// TwinCAT 3 PLC project SIM_1
// ProgramVersion: 3.1.4026.25
// libraries:
//   OC_Core, * (Open Commissioning)
//   Tc2_Math, * (Beckhoff Automation GmbH)
//   Tc2_Standard, * (Beckhoff Automation GmbH)
//   Tc2_System, * (Beckhoff Automation GmbH)
//   Tc2_Utilities, * (Beckhoff Automation GmbH)
//   Tc3_Module, * (Beckhoff Automation GmbH)
// project tree:
//   FG_01/ FG_01.TcPOU
//   FG_02/ FG_02.TcPOU
//   FG_03/ FG_03.TcPOU
//   FG_04/ FG_04.TcPOU
//   FG_05/ FG_05.TcPOU
//   FG_System/ FG_System.TcPOU
//   FG_Transport/ FG_Transport.TcPOU
//   Library/ FB_Camera.TcPOU
//   / MAIN.TcPOU (not stored), PlcTask.TcTTO
//   Sil/PLC/ GVL_PLC.TcGVL, ST_PLCInputs.TcDUT, ST_PLCOutputs.TcDUT
// real-time tasks:
//   TASK PlcTask: cycle T#1ms, priority 4, ADS port 350

CONFIGURATION SIM_1
    RESOURCE PLC ON TwinCAT3
        TASK PlcTask(INTERVAL := T#1ms, PRIORITY := 4);
        PROGRAM MAIN WITH PlcTask : MAIN;
    END_RESOURCE
END_CONFIGURATION

// ---- Sil/PLC/ST_PLCInputs.TcDUT
{attribute 'pack_mode' := '0'}
TYPE ST_PLCInputs :
STRUCT
	I0: BYTE;
	I1: BYTE;
	I2: BYTE;
	I3: BYTE;
	I4: BYTE;
	I5: BYTE;
	I6: BYTE;
	I7: BYTE;
	I8: BYTE;
	I9: BYTE;
	I10: BYTE;
	I11: BYTE;
	I12: BYTE;
	I13: BYTE;
	I14: BYTE;
	I15: BYTE;
	I16: BYTE;
	I17: BYTE;
	I18: BYTE;
	I19: BYTE;
	I20: BYTE;
	I21: BYTE;
	I22: BYTE;
	I23: BYTE;
	I24: BYTE;
	I25: BYTE;
	I26: BYTE;
	I27: BYTE;
	I28: BYTE;
	I29: BYTE;
	I30: BYTE;
	I31: BYTE;
	I32: BYTE;
	I33: BYTE;
	I34: BYTE;
	I35: BYTE;
	I36: BYTE;
	I37: BYTE;
	I38: BYTE;
	I39: BYTE;
	I40: BYTE;
	I41: BYTE;
	I42: BYTE;
	I43: BYTE;
	I44: BYTE;
	I45: BYTE;
	I46: BYTE;
	I47: BYTE;
	I48: BYTE;
	I49: BYTE;
	I50: BYTE;
	I51: BYTE;
	I52: BYTE;
	I53: BYTE;
	I54: BYTE;
	I55: BYTE;
	I56: BYTE;
	I57: BYTE;
	I58: BYTE;
	I59: BYTE;
	I60: BYTE;
	I61: BYTE;
	I62: BYTE;
	I63: BYTE;
	I64: BYTE;
	I65: BYTE;
	I66: BYTE;
	I67: BYTE;
	I68: BYTE;
	I69: BYTE;
	I70: BYTE;
	I71: BYTE;
	I72: BYTE;
	I73: BYTE;
	I74: BYTE;
	I75: BYTE;
	I76: BYTE;
	I77: BYTE;
	I78: BYTE;
	I79: BYTE;
	I80: BYTE;
	I81: BYTE;
	I82: BYTE;
	I83: BYTE;
	I84: BYTE;
	I85: BYTE;
	I86: BYTE;
	I87: BYTE;
	I88: BYTE;
	I89: BYTE;
	I90: BYTE;
	I91: BYTE;
	I92: BYTE;
	I93: BYTE;
	I94: BYTE;
	I95: BYTE;
	I96: BYTE;
	I97: BYTE;
	I98: BYTE;
	I99: BYTE;
	I100: BYTE;
	I101: BYTE;
	I102: BYTE;
	I103: BYTE;
	I104: BYTE;
	I105: BYTE;
	I106: BYTE;
	I107: BYTE;
	I108: BYTE;
	I109: BYTE;
	I110: BYTE;
	I111: BYTE;
	I112: BYTE;
	I113: BYTE;
	I114: BYTE;
	I115: BYTE;
	I116: BYTE;
	I117: BYTE;
	I118: BYTE;
	I119: BYTE;
	I120: BYTE;
	I121: BYTE;
	I122: BYTE;
	I123: BYTE;
	I124: BYTE;
	I125: BYTE;
	I126: BYTE;
	I127: BYTE;
	I128: BYTE;
	I129: BYTE;
	I130: BYTE;
	I131: BYTE;
	I132: BYTE;
	I133: BYTE;
	I134: BYTE;
	I135: BYTE;
	I136: BYTE;
	I137: BYTE;
	I138: BYTE;
	I139: BYTE;
	I140: BYTE;
	I141: BYTE;
	I142: BYTE;
	I143: BYTE;
	I144: BYTE;
	I145: BYTE;
	I146: BYTE;
	I147: BYTE;
	I148: BYTE;
	I149: BYTE;
	I150: BYTE;
	I151: BYTE;
	I152: BYTE;
	I153: BYTE;
	I154: BYTE;
	I155: BYTE;
	I156: BYTE;
	I157: BYTE;
	I158: BYTE;
	I159: BYTE;
	I160: BYTE;
	I161: BYTE;
	I162: BYTE;
	I163: BYTE;
	I164: BYTE;
	I165: BYTE;
	I166: BYTE;
	I167: BYTE;
	I168: BYTE;
	I169: BYTE;
	I170: BYTE;
	I171: BYTE;
	I172: BYTE;
	I173: BYTE;
	I174: BYTE;
	I175: BYTE;
	I176: BYTE;
	I177: BYTE;
	I178: BYTE;
	I179: BYTE;
	I180: BYTE;
	I181: BYTE;
	I182: BYTE;
	I183: BYTE;
	I184: BYTE;
	I185: BYTE;
	I186: BYTE;
	I187: BYTE;
	I188: BYTE;
	I189: BYTE;
	I190: BYTE;
	I191: BYTE;
	I192: BYTE;
	I193: BYTE;
	I194: BYTE;
	I195: BYTE;
	I196: BYTE;
	I197: BYTE;
	I198: BYTE;
	I199: BYTE;
	I200: BYTE;
	I201: BYTE;
	I202: BYTE;
	I203: BYTE;
	I204: BYTE;
	I205: BYTE;
	I206: BYTE;
	I207: BYTE;
	I208: BYTE;
	I209: BYTE;
	I210: BYTE;
	I211: BYTE;
	I212: BYTE;
	I213: BYTE;
	I214: BYTE;
	I215: BYTE;
	I216: BYTE;
	I217: BYTE;
	I218: BYTE;
	I219: BYTE;
	I220: BYTE;
	I221: BYTE;
	I222: BYTE;
	I223: BYTE;
	I224: BYTE;
	I225: BYTE;
	I226: BYTE;
	I227: BYTE;
	I228: BYTE;
	I229: BYTE;
	I230: BYTE;
	I231: BYTE;
	I232: BYTE;
	I233: BYTE;
	I234: BYTE;
	I235: BYTE;
	I236: BYTE;
	I237: BYTE;
	I238: BYTE;
	I239: BYTE;
	I240: BYTE;
	I241: BYTE;
	I242: BYTE;
	I243: BYTE;
	I244: BYTE;
	I245: BYTE;
	I246: BYTE;
	I247: BYTE;
	I248: BYTE;
	I249: BYTE;
	I250: BYTE;
	I251: BYTE;
	I252: BYTE;
	I253: BYTE;
	I254: BYTE;
	I255: BYTE;
	I256: BYTE;
	I257: BYTE;
	I258: BYTE;
	I259: BYTE;
	I260: BYTE;
	I261: BYTE;
	I262: BYTE;
	I263: BYTE;
	I264: BYTE;
	I265: BYTE;
	I266: BYTE;
	I267: BYTE;
	I268: BYTE;
	I269: BYTE;
	I270: BYTE;
	I271: BYTE;
	I272: BYTE;
	I273: BYTE;
	I274: BYTE;
	I275: BYTE;
	I276: BYTE;
	I277: BYTE;
	I278: BYTE;
	I279: BYTE;
	I280: BYTE;
	I281: BYTE;
	I282: BYTE;
	I283: BYTE;
	I284: BYTE;
	I285: BYTE;
	I286: BYTE;
	I287: BYTE;
	I288: BYTE;
	I289: BYTE;
	I290: BYTE;
	I291: BYTE;
	I292: BYTE;
	I293: BYTE;
	I294: BYTE;
	I295: BYTE;
	I296: BYTE;
	I297: BYTE;
	I298: BYTE;
	I299: BYTE;
	I300: BYTE;
	I301: BYTE;
	I302: BYTE;
	I303: BYTE;
	I304: BYTE;
	I305: BYTE;
	I306: BYTE;
	I307: BYTE;
	I308: BYTE;
	I309: BYTE;
	I310: BYTE;
	I311: BYTE;
	I312: BYTE;
	I313: BYTE;
	I314: BYTE;
	I315: BYTE;
	I316: BYTE;
	I317: BYTE;
	I318: BYTE;
	I319: BYTE;
	I320: BYTE;
	I321: BYTE;
	I322: BYTE;
	I323: BYTE;
	I324: BYTE;
	I325: BYTE;
	I326: BYTE;
	I327: BYTE;
	I328: BYTE;
	I329: BYTE;
	I330: BYTE;
	I331: BYTE;
	I332: BYTE;
	I333: BYTE;
	I334: BYTE;
	I335: BYTE;
	I336: BYTE;
	I337: BYTE;
	I338: BYTE;
	I339: BYTE;
	I340: BYTE;
	I341: BYTE;
	I342: BYTE;
	I343: BYTE;
	I344: BYTE;
	I345: BYTE;
	I346: BYTE;
	I347: BYTE;
	I348: BYTE;
	I349: BYTE;
	I350: BYTE;
	I351: BYTE;
	I352: BYTE;
	I353: BYTE;
	I354: BYTE;
	I355: BYTE;
	I356: BYTE;
	I357: BYTE;
	I358: BYTE;
	I359: BYTE;
	I360: BYTE;
	I361: BYTE;
	I362: BYTE;
	I363: BYTE;
	I364: BYTE;
	I365: BYTE;
	I366: BYTE;
	I367: BYTE;
	I368: BYTE;
	I369: BYTE;
	I370: BYTE;
	I371: BYTE;
	I372: BYTE;
	I373: BYTE;
	I374: BYTE;
	I375: BYTE;
	I376: BYTE;
	I377: BYTE;
	I378: BYTE;
	I379: BYTE;
	I380: BYTE;
	I381: BYTE;
	I382: BYTE;
	I383: BYTE;
	I384: BYTE;
	I385: BYTE;
	I386: BYTE;
	I387: BYTE;
	I388: BYTE;
	I389: BYTE;
	I390: BYTE;
	I391: BYTE;
	I392: BYTE;
	I393: BYTE;
	I394: BYTE;
	I395: BYTE;
	I396: BYTE;
	I397: BYTE;
	I398: BYTE;
	I399: BYTE;
	I400: BYTE;
	I401: BYTE;
	I402: BYTE;
	I403: BYTE;
	I404: BYTE;
	I405: BYTE;
	I406: BYTE;
	I407: BYTE;
	I408: BYTE;
	I409: BYTE;
	I410: BYTE;
	I411: BYTE;
	I412: BYTE;
	I413: BYTE;
	I414: BYTE;
	I415: BYTE;
	I416: BYTE;
	I417: BYTE;
	I418: BYTE;
	I419: BYTE;
	I420: BYTE;
	I421: BYTE;
	I422: BYTE;
	I423: BYTE;
	I424: BYTE;
	I425: BYTE;
	I426: BYTE;
	I427: BYTE;
	I428: BYTE;
	I429: BYTE;
	I430: BYTE;
	I431: BYTE;
	I432: BYTE;
	I433: BYTE;
	I434: BYTE;
	I435: BYTE;
	I436: BYTE;
	I437: BYTE;
	I438: BYTE;
	I439: BYTE;
	I440: BYTE;
	I441: BYTE;
	I442: BYTE;
	I443: BYTE;
	I444: BYTE;
	I445: BYTE;
	I446: BYTE;
	I447: BYTE;
	I448: BYTE;
	I449: BYTE;
	I450: BYTE;
	I451: BYTE;
	I452: BYTE;
	I453: BYTE;
	I454: BYTE;
	I455: BYTE;
	I456: BYTE;
	I457: BYTE;
	I458: BYTE;
	I459: BYTE;
	I460: BYTE;
	I461: BYTE;
	I462: BYTE;
	I463: BYTE;
	I464: BYTE;
	I465: BYTE;
	I466: BYTE;
	I467: BYTE;
	I468: BYTE;
	I469: BYTE;
	I470: BYTE;
	I471: BYTE;
	I472: BYTE;
	I473: BYTE;
	I474: BYTE;
	I475: BYTE;
	I476: BYTE;
	I477: BYTE;
	I478: BYTE;
	I479: BYTE;
	I480: BYTE;
	I481: BYTE;
	I482: BYTE;
	I483: BYTE;
	I484: BYTE;
	I485: BYTE;
	I486: BYTE;
	I487: BYTE;
	I488: BYTE;
	I489: BYTE;
	I490: BYTE;
	I491: BYTE;
	I492: BYTE;
	I493: BYTE;
	I494: BYTE;
	I495: BYTE;
	I496: BYTE;
	I497: BYTE;
	I498: BYTE;
	I499: BYTE;
	I500: BYTE;
	I501: BYTE;
	I502: BYTE;
	I503: BYTE;
	I504: BYTE;
	I505: BYTE;
	I506: BYTE;
	I507: BYTE;
	I508: BYTE;
	I509: BYTE;
	I510: BYTE;
	I511: BYTE;
	I512: BYTE;
	I513: BYTE;
	I514: BYTE;
	I515: BYTE;
	I516: BYTE;
	I517: BYTE;
	I518: BYTE;
	I519: BYTE;
	I520: BYTE;
	I521: BYTE;
	I522: BYTE;
	I523: BYTE;
	I524: BYTE;
	I525: BYTE;
	I526: BYTE;
	I527: BYTE;
	I528: BYTE;
	I529: BYTE;
	I530: BYTE;
	I531: BYTE;
	I532: BYTE;
	I533: BYTE;
	I534: BYTE;
	I535: BYTE;
	I536: BYTE;
	I537: BYTE;
	I538: BYTE;
	I539: BYTE;
	I540: BYTE;
	I541: BYTE;
	I542: BYTE;
	I543: BYTE;
	I544: BYTE;
	I545: BYTE;
	I546: BYTE;
	I547: BYTE;
	I548: BYTE;
	I549: BYTE;
	I550: BYTE;
	I551: BYTE;
	I552: BYTE;
	I553: BYTE;
	I554: BYTE;
	I555: BYTE;
	I556: BYTE;
	I557: BYTE;
	I558: BYTE;
	I559: BYTE;
	I560: BYTE;
	I561: BYTE;
	I562: BYTE;
	I563: BYTE;
	I564: BYTE;
	I565: BYTE;
	I566: BYTE;
	I567: BYTE;
	I568: BYTE;
	I569: BYTE;
	I570: BYTE;
	I571: BYTE;
	I572: BYTE;
	I573: BYTE;
	I574: BYTE;
	I575: BYTE;
	I576: BYTE;
	I577: BYTE;
	I578: BYTE;
	I579: BYTE;
	I580: BYTE;
	I581: BYTE;
	I582: BYTE;
	I583: BYTE;
	I584: BYTE;
	I585: BYTE;
	I586: BYTE;
	I587: BYTE;
	I588: BYTE;
	I589: BYTE;
	I590: BYTE;
	I591: BYTE;
	I592: BYTE;
	I593: BYTE;
	I594: BYTE;
	I595: BYTE;
	I596: BYTE;
	I597: BYTE;
	I598: BYTE;
	I599: BYTE;
	I600: BYTE;
	I601: BYTE;
	I602: BYTE;
	I603: BYTE;
	I604: BYTE;
	I605: BYTE;
	I606: BYTE;
	I607: BYTE;
	I608: BYTE;
	I609: BYTE;
	I610: BYTE;
	I611: BYTE;
	I612: BYTE;
	I613: BYTE;
	I614: BYTE;
	I615: BYTE;
	I616: BYTE;
	I617: BYTE;
	I618: BYTE;
	I619: BYTE;
	I620: BYTE;
	I621: BYTE;
	I622: BYTE;
	I623: BYTE;
	I624: BYTE;
	I625: BYTE;
	I626: BYTE;
	I627: BYTE;
	I628: BYTE;
	I629: BYTE;
	I630: BYTE;
	I631: BYTE;
	I632: BYTE;
	I633: BYTE;
	I634: BYTE;
	I635: BYTE;
	I636: BYTE;
	I637: BYTE;
	I638: BYTE;
	I639: BYTE;
	I640: BYTE;
	I641: BYTE;
	I642: BYTE;
	I643: BYTE;
	I644: BYTE;
	I645: BYTE;
	I646: BYTE;
	I647: BYTE;
	I648: BYTE;
	I649: BYTE;
	I650: BYTE;
	I651: BYTE;
	I652: BYTE;
	I653: BYTE;
	I654: BYTE;
	I655: BYTE;
	I656: BYTE;
	I657: BYTE;
	I658: BYTE;
	I659: BYTE;
	I660: BYTE;
	I661: BYTE;
	I662: BYTE;
	I663: BYTE;
	I664: BYTE;
	I665: BYTE;
	I666: BYTE;
	I667: BYTE;
	I668: BYTE;
	I669: BYTE;
	I670: BYTE;
	I671: BYTE;
	I672: BYTE;
	I673: BYTE;
	I674: BYTE;
	I675: BYTE;
	I676: BYTE;
	I677: BYTE;
	I678: BYTE;
	I679: BYTE;
	I680: BYTE;
	I681: BYTE;
	I682: BYTE;
	I683: BYTE;
	I684: BYTE;
	I685: BYTE;
	I686: BYTE;
	I687: BYTE;
	I688: BYTE;
	I689: BYTE;
	I690: BYTE;
	I691: BYTE;
	I692: BYTE;
	I693: BYTE;
	I694: BYTE;
	I695: BYTE;
	I696: BYTE;
	I697: BYTE;
	I698: BYTE;
	I699: BYTE;
	I700: BYTE;
	I701: BYTE;
	I702: BYTE;
	I703: BYTE;
	I704: BYTE;
	I705: BYTE;
	I706: BYTE;
	I707: BYTE;
	I708: BYTE;
	I709: BYTE;
	I710: BYTE;
	I711: BYTE;
	I712: BYTE;
	I713: BYTE;
	I714: BYTE;
	I715: BYTE;
	I716: BYTE;
	I717: BYTE;
	I718: BYTE;
	I719: BYTE;
	I720: BYTE;
	I721: BYTE;
	I722: BYTE;
	I723: BYTE;
	I724: BYTE;
	I725: BYTE;
	I726: BYTE;
	I727: BYTE;
	I728: BYTE;
	I729: BYTE;
	I730: BYTE;
	I731: BYTE;
	I732: BYTE;
	I733: BYTE;
	I734: BYTE;
	I735: BYTE;
	I736: BYTE;
	I737: BYTE;
	I738: BYTE;
	I739: BYTE;
	I740: BYTE;
	I741: BYTE;
	I742: BYTE;
	I743: BYTE;
	I744: BYTE;
	I745: BYTE;
	I746: BYTE;
	I747: BYTE;
	I748: BYTE;
	I749: BYTE;
	I750: BYTE;
	I751: BYTE;
	I752: BYTE;
	I753: BYTE;
	I754: BYTE;
	I755: BYTE;
	I756: BYTE;
	I757: BYTE;
	I758: BYTE;
	I759: BYTE;
	I760: BYTE;
	I761: BYTE;
	I762: BYTE;
	I763: BYTE;
	I764: BYTE;
	I765: BYTE;
	I766: BYTE;
	I767: BYTE;
	I768: BYTE;
	I769: BYTE;
	I770: BYTE;
	I771: BYTE;
	I772: BYTE;
	I773: BYTE;
	I774: BYTE;
	I775: BYTE;
	I776: BYTE;
	I777: BYTE;
	I778: BYTE;
	I779: BYTE;
	I780: BYTE;
	I781: BYTE;
	I782: BYTE;
	I783: BYTE;
	I784: BYTE;
	I785: BYTE;
	I786: BYTE;
	I787: BYTE;
	I788: BYTE;
	I789: BYTE;
	I790: BYTE;
	I791: BYTE;
	I792: BYTE;
	I793: BYTE;
	I794: BYTE;
	I795: BYTE;
	I796: BYTE;
	I797: BYTE;
	I798: BYTE;
	I799: BYTE;
	I800: BYTE;
	I801: BYTE;
	I802: BYTE;
	I803: BYTE;
	I804: BYTE;
	I805: BYTE;
	I806: BYTE;
	I807: BYTE;
	I808: BYTE;
	I809: BYTE;
	I810: BYTE;
	I811: BYTE;
	I812: BYTE;
	I813: BYTE;
	I814: BYTE;
	I815: BYTE;
	I816: BYTE;
	I817: BYTE;
	I818: BYTE;
	I819: BYTE;
	I820: BYTE;
	I821: BYTE;
	I822: BYTE;
	I823: BYTE;
	I824: BYTE;
	I825: BYTE;
	I826: BYTE;
	I827: BYTE;
	I828: BYTE;
	I829: BYTE;
	I830: BYTE;
	I831: BYTE;
	I832: BYTE;
	I833: BYTE;
	I834: BYTE;
	I835: BYTE;
	I836: BYTE;
	I837: BYTE;
	I838: BYTE;
	I839: BYTE;
	I840: BYTE;
	I841: BYTE;
	I842: BYTE;
	I843: BYTE;
	I844: BYTE;
	I845: BYTE;
	I846: BYTE;
	I847: BYTE;
	I848: BYTE;
	I849: BYTE;
	I850: BYTE;
	I851: BYTE;
	I852: BYTE;
	I853: BYTE;
	I854: BYTE;
	I855: BYTE;
	I856: BYTE;
	I857: BYTE;
	I858: BYTE;
	I859: BYTE;
	I860: BYTE;
	I861: BYTE;
	I862: BYTE;
	I863: BYTE;
	I864: BYTE;
	I865: BYTE;
	I866: BYTE;
	I867: BYTE;
	I868: BYTE;
	I869: BYTE;
	I870: BYTE;
	I871: BYTE;
	I872: BYTE;
	I873: BYTE;
	I874: BYTE;
	I875: BYTE;
	I876: BYTE;
	I877: BYTE;
	I878: BYTE;
	I879: BYTE;
	I880: BYTE;
	I881: BYTE;
	I882: BYTE;
	I883: BYTE;
	I884: BYTE;
	I885: BYTE;
	I886: BYTE;
	I887: BYTE;
	I888: BYTE;
	I889: BYTE;
	I890: BYTE;
	I891: BYTE;
	I892: BYTE;
	I893: BYTE;
	I894: BYTE;
	I895: BYTE;
	I896: BYTE;
	I897: BYTE;
	I898: BYTE;
	I899: BYTE;
	I900: BYTE;
	I901: BYTE;
	I902: BYTE;
	I903: BYTE;
	I904: BYTE;
	I905: BYTE;
	I906: BYTE;
	I907: BYTE;
	I908: BYTE;
	I909: BYTE;
	I910: BYTE;
	I911: BYTE;
	I912: BYTE;
	I913: BYTE;
	I914: BYTE;
	I915: BYTE;
	I916: BYTE;
	I917: BYTE;
	I918: BYTE;
	I919: BYTE;
	I920: BYTE;
	I921: BYTE;
	I922: BYTE;
	I923: BYTE;
	I924: BYTE;
	I925: BYTE;
	I926: BYTE;
	I927: BYTE;
	I928: BYTE;
	I929: BYTE;
	I930: BYTE;
	I931: BYTE;
	I932: BYTE;
	I933: BYTE;
	I934: BYTE;
	I935: BYTE;
	I936: BYTE;
	I937: BYTE;
	I938: BYTE;
	I939: BYTE;
	I940: BYTE;
	I941: BYTE;
	I942: BYTE;
	I943: BYTE;
	I944: BYTE;
	I945: BYTE;
	I946: BYTE;
	I947: BYTE;
	I948: BYTE;
	I949: BYTE;
	I950: BYTE;
	I951: BYTE;
	I952: BYTE;
	I953: BYTE;
	I954: BYTE;
	I955: BYTE;
	I956: BYTE;
	I957: BYTE;
	I958: BYTE;
	I959: BYTE;
	I960: BYTE;
	I961: BYTE;
	I962: BYTE;
	I963: BYTE;
	I964: BYTE;
	I965: BYTE;
	I966: BYTE;
	I967: BYTE;
	I968: BYTE;
	I969: BYTE;
	I970: BYTE;
	I971: BYTE;
	I972: BYTE;
	I973: BYTE;
	I974: BYTE;
	I975: BYTE;
	I976: BYTE;
	I977: BYTE;
	I978: BYTE;
	I979: BYTE;
	I980: BYTE;
	I981: BYTE;
	I982: BYTE;
	I983: BYTE;
	I984: BYTE;
	I985: BYTE;
	I986: BYTE;
	I987: BYTE;
	I988: BYTE;
	I989: BYTE;
	I990: BYTE;
	I991: BYTE;
	I992: BYTE;
	I993: BYTE;
	I994: BYTE;
	I995: BYTE;
	I996: BYTE;
	I997: BYTE;
	I998: BYTE;
	I999: BYTE;
	I1000: BYTE;
	I1001: BYTE;
	I1002: BYTE;
	I1003: BYTE;
	I1004: BYTE;
	I1005: BYTE;
	I1006: BYTE;
	I1007: BYTE;
	I1008: BYTE;
	I1009: BYTE;
	I1010: BYTE;
	I1011: BYTE;
	I1012: BYTE;
	I1013: BYTE;
	I1014: BYTE;
	I1015: BYTE;
	I1016: BYTE;
	I1017: BYTE;
	I1018: BYTE;
	I1019: BYTE;
	I1020: BYTE;
	I1021: BYTE;
	I1022: BYTE;
	I1023: BYTE;
END_STRUCT
END_TYPE

// ---- Sil/PLC/ST_PLCOutputs.TcDUT
{attribute 'pack_mode' := '0'}
TYPE ST_PLCOutputs :
STRUCT
	Q0: BYTE;
	Q1: BYTE;
	Q2: BYTE;
	Q3: BYTE;
	Q4: BYTE;
	Q5: BYTE;
	Q6: BYTE;
	Q7: BYTE;
	Q8: BYTE;
	Q9: BYTE;
	Q10: BYTE;
	Q11: BYTE;
	Q12: BYTE;
	Q13: BYTE;
	Q14: BYTE;
	Q15: BYTE;
	Q16: BYTE;
	Q17: BYTE;
	Q18: BYTE;
	Q19: BYTE;
	Q20: BYTE;
	Q21: BYTE;
	Q22: BYTE;
	Q23: BYTE;
	Q24: BYTE;
	Q25: BYTE;
	Q26: BYTE;
	Q27: BYTE;
	Q28: BYTE;
	Q29: BYTE;
	Q30: BYTE;
	Q31: BYTE;
	Q32: BYTE;
	Q33: BYTE;
	Q34: BYTE;
	Q35: BYTE;
	Q36: BYTE;
	Q37: BYTE;
	Q38: BYTE;
	Q39: BYTE;
	Q40: BYTE;
	Q41: BYTE;
	Q42: BYTE;
	Q43: BYTE;
	Q44: BYTE;
	Q45: BYTE;
	Q46: BYTE;
	Q47: BYTE;
	Q48: BYTE;
	Q49: BYTE;
	Q50: BYTE;
	Q51: BYTE;
	Q52: BYTE;
	Q53: BYTE;
	Q54: BYTE;
	Q55: BYTE;
	Q56: BYTE;
	Q57: BYTE;
	Q58: BYTE;
	Q59: BYTE;
	Q60: BYTE;
	Q61: BYTE;
	Q62: BYTE;
	Q63: BYTE;
	Q64: BYTE;
	Q65: BYTE;
	Q66: BYTE;
	Q67: BYTE;
	Q68: BYTE;
	Q69: BYTE;
	Q70: BYTE;
	Q71: BYTE;
	Q72: BYTE;
	Q73: BYTE;
	Q74: BYTE;
	Q75: BYTE;
	Q76: BYTE;
	Q77: BYTE;
	Q78: BYTE;
	Q79: BYTE;
	Q80: BYTE;
	Q81: BYTE;
	Q82: BYTE;
	Q83: BYTE;
	Q84: BYTE;
	Q85: BYTE;
	Q86: BYTE;
	Q87: BYTE;
	Q88: BYTE;
	Q89: BYTE;
	Q90: BYTE;
	Q91: BYTE;
	Q92: BYTE;
	Q93: BYTE;
	Q94: BYTE;
	Q95: BYTE;
	Q96: BYTE;
	Q97: BYTE;
	Q98: BYTE;
	Q99: BYTE;
	Q100: BYTE;
	Q101: BYTE;
	Q102: BYTE;
	Q103: BYTE;
	Q104: BYTE;
	Q105: BYTE;
	Q106: BYTE;
	Q107: BYTE;
	Q108: BYTE;
	Q109: BYTE;
	Q110: BYTE;
	Q111: BYTE;
	Q112: BYTE;
	Q113: BYTE;
	Q114: BYTE;
	Q115: BYTE;
	Q116: BYTE;
	Q117: BYTE;
	Q118: BYTE;
	Q119: BYTE;
	Q120: BYTE;
	Q121: BYTE;
	Q122: BYTE;
	Q123: BYTE;
	Q124: BYTE;
	Q125: BYTE;
	Q126: BYTE;
	Q127: BYTE;
	Q128: BYTE;
	Q129: BYTE;
	Q130: BYTE;
	Q131: BYTE;
	Q132: BYTE;
	Q133: BYTE;
	Q134: BYTE;
	Q135: BYTE;
	Q136: BYTE;
	Q137: BYTE;
	Q138: BYTE;
	Q139: BYTE;
	Q140: BYTE;
	Q141: BYTE;
	Q142: BYTE;
	Q143: BYTE;
	Q144: BYTE;
	Q145: BYTE;
	Q146: BYTE;
	Q147: BYTE;
	Q148: BYTE;
	Q149: BYTE;
	Q150: BYTE;
	Q151: BYTE;
	Q152: BYTE;
	Q153: BYTE;
	Q154: BYTE;
	Q155: BYTE;
	Q156: BYTE;
	Q157: BYTE;
	Q158: BYTE;
	Q159: BYTE;
	Q160: BYTE;
	Q161: BYTE;
	Q162: BYTE;
	Q163: BYTE;
	Q164: BYTE;
	Q165: BYTE;
	Q166: BYTE;
	Q167: BYTE;
	Q168: BYTE;
	Q169: BYTE;
	Q170: BYTE;
	Q171: BYTE;
	Q172: BYTE;
	Q173: BYTE;
	Q174: BYTE;
	Q175: BYTE;
	Q176: BYTE;
	Q177: BYTE;
	Q178: BYTE;
	Q179: BYTE;
	Q180: BYTE;
	Q181: BYTE;
	Q182: BYTE;
	Q183: BYTE;
	Q184: BYTE;
	Q185: BYTE;
	Q186: BYTE;
	Q187: BYTE;
	Q188: BYTE;
	Q189: BYTE;
	Q190: BYTE;
	Q191: BYTE;
	Q192: BYTE;
	Q193: BYTE;
	Q194: BYTE;
	Q195: BYTE;
	Q196: BYTE;
	Q197: BYTE;
	Q198: BYTE;
	Q199: BYTE;
	Q200: BYTE;
	Q201: BYTE;
	Q202: BYTE;
	Q203: BYTE;
	Q204: BYTE;
	Q205: BYTE;
	Q206: BYTE;
	Q207: BYTE;
	Q208: BYTE;
	Q209: BYTE;
	Q210: BYTE;
	Q211: BYTE;
	Q212: BYTE;
	Q213: BYTE;
	Q214: BYTE;
	Q215: BYTE;
	Q216: BYTE;
	Q217: BYTE;
	Q218: BYTE;
	Q219: BYTE;
	Q220: BYTE;
	Q221: BYTE;
	Q222: BYTE;
	Q223: BYTE;
	Q224: BYTE;
	Q225: BYTE;
	Q226: BYTE;
	Q227: BYTE;
	Q228: BYTE;
	Q229: BYTE;
	Q230: BYTE;
	Q231: BYTE;
	Q232: BYTE;
	Q233: BYTE;
	Q234: BYTE;
	Q235: BYTE;
	Q236: BYTE;
	Q237: BYTE;
	Q238: BYTE;
	Q239: BYTE;
	Q240: BYTE;
	Q241: BYTE;
	Q242: BYTE;
	Q243: BYTE;
	Q244: BYTE;
	Q245: BYTE;
	Q246: BYTE;
	Q247: BYTE;
	Q248: BYTE;
	Q249: BYTE;
	Q250: BYTE;
	Q251: BYTE;
	Q252: BYTE;
	Q253: BYTE;
	Q254: BYTE;
	Q255: BYTE;
	Q256: BYTE;
	Q257: BYTE;
	Q258: BYTE;
	Q259: BYTE;
	Q260: BYTE;
	Q261: BYTE;
	Q262: BYTE;
	Q263: BYTE;
	Q264: BYTE;
	Q265: BYTE;
	Q266: BYTE;
	Q267: BYTE;
	Q268: BYTE;
	Q269: BYTE;
	Q270: BYTE;
	Q271: BYTE;
	Q272: BYTE;
	Q273: BYTE;
	Q274: BYTE;
	Q275: BYTE;
	Q276: BYTE;
	Q277: BYTE;
	Q278: BYTE;
	Q279: BYTE;
	Q280: BYTE;
	Q281: BYTE;
	Q282: BYTE;
	Q283: BYTE;
	Q284: BYTE;
	Q285: BYTE;
	Q286: BYTE;
	Q287: BYTE;
	Q288: BYTE;
	Q289: BYTE;
	Q290: BYTE;
	Q291: BYTE;
	Q292: BYTE;
	Q293: BYTE;
	Q294: BYTE;
	Q295: BYTE;
	Q296: BYTE;
	Q297: BYTE;
	Q298: BYTE;
	Q299: BYTE;
	Q300: BYTE;
	Q301: BYTE;
	Q302: BYTE;
	Q303: BYTE;
	Q304: BYTE;
	Q305: BYTE;
	Q306: BYTE;
	Q307: BYTE;
	Q308: BYTE;
	Q309: BYTE;
	Q310: BYTE;
	Q311: BYTE;
	Q312: BYTE;
	Q313: BYTE;
	Q314: BYTE;
	Q315: BYTE;
	Q316: BYTE;
	Q317: BYTE;
	Q318: BYTE;
	Q319: BYTE;
	Q320: BYTE;
	Q321: BYTE;
	Q322: BYTE;
	Q323: BYTE;
	Q324: BYTE;
	Q325: BYTE;
	Q326: BYTE;
	Q327: BYTE;
	Q328: BYTE;
	Q329: BYTE;
	Q330: BYTE;
	Q331: BYTE;
	Q332: BYTE;
	Q333: BYTE;
	Q334: BYTE;
	Q335: BYTE;
	Q336: BYTE;
	Q337: BYTE;
	Q338: BYTE;
	Q339: BYTE;
	Q340: BYTE;
	Q341: BYTE;
	Q342: BYTE;
	Q343: BYTE;
	Q344: BYTE;
	Q345: BYTE;
	Q346: BYTE;
	Q347: BYTE;
	Q348: BYTE;
	Q349: BYTE;
	Q350: BYTE;
	Q351: BYTE;
	Q352: BYTE;
	Q353: BYTE;
	Q354: BYTE;
	Q355: BYTE;
	Q356: BYTE;
	Q357: BYTE;
	Q358: BYTE;
	Q359: BYTE;
	Q360: BYTE;
	Q361: BYTE;
	Q362: BYTE;
	Q363: BYTE;
	Q364: BYTE;
	Q365: BYTE;
	Q366: BYTE;
	Q367: BYTE;
	Q368: BYTE;
	Q369: BYTE;
	Q370: BYTE;
	Q371: BYTE;
	Q372: BYTE;
	Q373: BYTE;
	Q374: BYTE;
	Q375: BYTE;
	Q376: BYTE;
	Q377: BYTE;
	Q378: BYTE;
	Q379: BYTE;
	Q380: BYTE;
	Q381: BYTE;
	Q382: BYTE;
	Q383: BYTE;
	Q384: BYTE;
	Q385: BYTE;
	Q386: BYTE;
	Q387: BYTE;
	Q388: BYTE;
	Q389: BYTE;
	Q390: BYTE;
	Q391: BYTE;
	Q392: BYTE;
	Q393: BYTE;
	Q394: BYTE;
	Q395: BYTE;
	Q396: BYTE;
	Q397: BYTE;
	Q398: BYTE;
	Q399: BYTE;
	Q400: BYTE;
	Q401: BYTE;
	Q402: BYTE;
	Q403: BYTE;
	Q404: BYTE;
	Q405: BYTE;
	Q406: BYTE;
	Q407: BYTE;
	Q408: BYTE;
	Q409: BYTE;
	Q410: BYTE;
	Q411: BYTE;
	Q412: BYTE;
	Q413: BYTE;
	Q414: BYTE;
	Q415: BYTE;
	Q416: BYTE;
	Q417: BYTE;
	Q418: BYTE;
	Q419: BYTE;
	Q420: BYTE;
	Q421: BYTE;
	Q422: BYTE;
	Q423: BYTE;
	Q424: BYTE;
	Q425: BYTE;
	Q426: BYTE;
	Q427: BYTE;
	Q428: BYTE;
	Q429: BYTE;
	Q430: BYTE;
	Q431: BYTE;
	Q432: BYTE;
	Q433: BYTE;
	Q434: BYTE;
	Q435: BYTE;
	Q436: BYTE;
	Q437: BYTE;
	Q438: BYTE;
	Q439: BYTE;
	Q440: BYTE;
	Q441: BYTE;
	Q442: BYTE;
	Q443: BYTE;
	Q444: BYTE;
	Q445: BYTE;
	Q446: BYTE;
	Q447: BYTE;
	Q448: BYTE;
	Q449: BYTE;
	Q450: BYTE;
	Q451: BYTE;
	Q452: BYTE;
	Q453: BYTE;
	Q454: BYTE;
	Q455: BYTE;
	Q456: BYTE;
	Q457: BYTE;
	Q458: BYTE;
	Q459: BYTE;
	Q460: BYTE;
	Q461: BYTE;
	Q462: BYTE;
	Q463: BYTE;
	Q464: BYTE;
	Q465: BYTE;
	Q466: BYTE;
	Q467: BYTE;
	Q468: BYTE;
	Q469: BYTE;
	Q470: BYTE;
	Q471: BYTE;
	Q472: BYTE;
	Q473: BYTE;
	Q474: BYTE;
	Q475: BYTE;
	Q476: BYTE;
	Q477: BYTE;
	Q478: BYTE;
	Q479: BYTE;
	Q480: BYTE;
	Q481: BYTE;
	Q482: BYTE;
	Q483: BYTE;
	Q484: BYTE;
	Q485: BYTE;
	Q486: BYTE;
	Q487: BYTE;
	Q488: BYTE;
	Q489: BYTE;
	Q490: BYTE;
	Q491: BYTE;
	Q492: BYTE;
	Q493: BYTE;
	Q494: BYTE;
	Q495: BYTE;
	Q496: BYTE;
	Q497: BYTE;
	Q498: BYTE;
	Q499: BYTE;
	Q500: BYTE;
	Q501: BYTE;
	Q502: BYTE;
	Q503: BYTE;
	Q504: BYTE;
	Q505: BYTE;
	Q506: BYTE;
	Q507: BYTE;
	Q508: BYTE;
	Q509: BYTE;
	Q510: BYTE;
	Q511: BYTE;
	Q512: BYTE;
	Q513: BYTE;
	Q514: BYTE;
	Q515: BYTE;
	Q516: BYTE;
	Q517: BYTE;
	Q518: BYTE;
	Q519: BYTE;
	Q520: BYTE;
	Q521: BYTE;
	Q522: BYTE;
	Q523: BYTE;
	Q524: BYTE;
	Q525: BYTE;
	Q526: BYTE;
	Q527: BYTE;
	Q528: BYTE;
	Q529: BYTE;
	Q530: BYTE;
	Q531: BYTE;
	Q532: BYTE;
	Q533: BYTE;
	Q534: BYTE;
	Q535: BYTE;
	Q536: BYTE;
	Q537: BYTE;
	Q538: BYTE;
	Q539: BYTE;
	Q540: BYTE;
	Q541: BYTE;
	Q542: BYTE;
	Q543: BYTE;
	Q544: BYTE;
	Q545: BYTE;
	Q546: BYTE;
	Q547: BYTE;
	Q548: BYTE;
	Q549: BYTE;
	Q550: BYTE;
	Q551: BYTE;
	Q552: BYTE;
	Q553: BYTE;
	Q554: BYTE;
	Q555: BYTE;
	Q556: BYTE;
	Q557: BYTE;
	Q558: BYTE;
	Q559: BYTE;
	Q560: BYTE;
	Q561: BYTE;
	Q562: BYTE;
	Q563: BYTE;
	Q564: BYTE;
	Q565: BYTE;
	Q566: BYTE;
	Q567: BYTE;
	Q568: BYTE;
	Q569: BYTE;
	Q570: BYTE;
	Q571: BYTE;
	Q572: BYTE;
	Q573: BYTE;
	Q574: BYTE;
	Q575: BYTE;
	Q576: BYTE;
	Q577: BYTE;
	Q578: BYTE;
	Q579: BYTE;
	Q580: BYTE;
	Q581: BYTE;
	Q582: BYTE;
	Q583: BYTE;
	Q584: BYTE;
	Q585: BYTE;
	Q586: BYTE;
	Q587: BYTE;
	Q588: BYTE;
	Q589: BYTE;
	Q590: BYTE;
	Q591: BYTE;
	Q592: BYTE;
	Q593: BYTE;
	Q594: BYTE;
	Q595: BYTE;
	Q596: BYTE;
	Q597: BYTE;
	Q598: BYTE;
	Q599: BYTE;
	Q600: BYTE;
	Q601: BYTE;
	Q602: BYTE;
	Q603: BYTE;
	Q604: BYTE;
	Q605: BYTE;
	Q606: BYTE;
	Q607: BYTE;
	Q608: BYTE;
	Q609: BYTE;
	Q610: BYTE;
	Q611: BYTE;
	Q612: BYTE;
	Q613: BYTE;
	Q614: BYTE;
	Q615: BYTE;
	Q616: BYTE;
	Q617: BYTE;
	Q618: BYTE;
	Q619: BYTE;
	Q620: BYTE;
	Q621: BYTE;
	Q622: BYTE;
	Q623: BYTE;
	Q624: BYTE;
	Q625: BYTE;
	Q626: BYTE;
	Q627: BYTE;
	Q628: BYTE;
	Q629: BYTE;
	Q630: BYTE;
	Q631: BYTE;
	Q632: BYTE;
	Q633: BYTE;
	Q634: BYTE;
	Q635: BYTE;
	Q636: BYTE;
	Q637: BYTE;
	Q638: BYTE;
	Q639: BYTE;
	Q640: BYTE;
	Q641: BYTE;
	Q642: BYTE;
	Q643: BYTE;
	Q644: BYTE;
	Q645: BYTE;
	Q646: BYTE;
	Q647: BYTE;
	Q648: BYTE;
	Q649: BYTE;
	Q650: BYTE;
	Q651: BYTE;
	Q652: BYTE;
	Q653: BYTE;
	Q654: BYTE;
	Q655: BYTE;
	Q656: BYTE;
	Q657: BYTE;
	Q658: BYTE;
	Q659: BYTE;
	Q660: BYTE;
	Q661: BYTE;
	Q662: BYTE;
	Q663: BYTE;
	Q664: BYTE;
	Q665: BYTE;
	Q666: BYTE;
	Q667: BYTE;
	Q668: BYTE;
	Q669: BYTE;
	Q670: BYTE;
	Q671: BYTE;
	Q672: BYTE;
	Q673: BYTE;
	Q674: BYTE;
	Q675: BYTE;
	Q676: BYTE;
	Q677: BYTE;
	Q678: BYTE;
	Q679: BYTE;
	Q680: BYTE;
	Q681: BYTE;
	Q682: BYTE;
	Q683: BYTE;
	Q684: BYTE;
	Q685: BYTE;
	Q686: BYTE;
	Q687: BYTE;
	Q688: BYTE;
	Q689: BYTE;
	Q690: BYTE;
	Q691: BYTE;
	Q692: BYTE;
	Q693: BYTE;
	Q694: BYTE;
	Q695: BYTE;
	Q696: BYTE;
	Q697: BYTE;
	Q698: BYTE;
	Q699: BYTE;
	Q700: BYTE;
	Q701: BYTE;
	Q702: BYTE;
	Q703: BYTE;
	Q704: BYTE;
	Q705: BYTE;
	Q706: BYTE;
	Q707: BYTE;
	Q708: BYTE;
	Q709: BYTE;
	Q710: BYTE;
	Q711: BYTE;
	Q712: BYTE;
	Q713: BYTE;
	Q714: BYTE;
	Q715: BYTE;
	Q716: BYTE;
	Q717: BYTE;
	Q718: BYTE;
	Q719: BYTE;
	Q720: BYTE;
	Q721: BYTE;
	Q722: BYTE;
	Q723: BYTE;
	Q724: BYTE;
	Q725: BYTE;
	Q726: BYTE;
	Q727: BYTE;
	Q728: BYTE;
	Q729: BYTE;
	Q730: BYTE;
	Q731: BYTE;
	Q732: BYTE;
	Q733: BYTE;
	Q734: BYTE;
	Q735: BYTE;
	Q736: BYTE;
	Q737: BYTE;
	Q738: BYTE;
	Q739: BYTE;
	Q740: BYTE;
	Q741: BYTE;
	Q742: BYTE;
	Q743: BYTE;
	Q744: BYTE;
	Q745: BYTE;
	Q746: BYTE;
	Q747: BYTE;
	Q748: BYTE;
	Q749: BYTE;
	Q750: BYTE;
	Q751: BYTE;
	Q752: BYTE;
	Q753: BYTE;
	Q754: BYTE;
	Q755: BYTE;
	Q756: BYTE;
	Q757: BYTE;
	Q758: BYTE;
	Q759: BYTE;
	Q760: BYTE;
	Q761: BYTE;
	Q762: BYTE;
	Q763: BYTE;
	Q764: BYTE;
	Q765: BYTE;
	Q766: BYTE;
	Q767: BYTE;
	Q768: BYTE;
	Q769: BYTE;
	Q770: BYTE;
	Q771: BYTE;
	Q772: BYTE;
	Q773: BYTE;
	Q774: BYTE;
	Q775: BYTE;
	Q776: BYTE;
	Q777: BYTE;
	Q778: BYTE;
	Q779: BYTE;
	Q780: BYTE;
	Q781: BYTE;
	Q782: BYTE;
	Q783: BYTE;
	Q784: BYTE;
	Q785: BYTE;
	Q786: BYTE;
	Q787: BYTE;
	Q788: BYTE;
	Q789: BYTE;
	Q790: BYTE;
	Q791: BYTE;
	Q792: BYTE;
	Q793: BYTE;
	Q794: BYTE;
	Q795: BYTE;
	Q796: BYTE;
	Q797: BYTE;
	Q798: BYTE;
	Q799: BYTE;
	Q800: BYTE;
	Q801: BYTE;
	Q802: BYTE;
	Q803: BYTE;
	Q804: BYTE;
	Q805: BYTE;
	Q806: BYTE;
	Q807: BYTE;
	Q808: BYTE;
	Q809: BYTE;
	Q810: BYTE;
	Q811: BYTE;
	Q812: BYTE;
	Q813: BYTE;
	Q814: BYTE;
	Q815: BYTE;
	Q816: BYTE;
	Q817: BYTE;
	Q818: BYTE;
	Q819: BYTE;
	Q820: BYTE;
	Q821: BYTE;
	Q822: BYTE;
	Q823: BYTE;
	Q824: BYTE;
	Q825: BYTE;
	Q826: BYTE;
	Q827: BYTE;
	Q828: BYTE;
	Q829: BYTE;
	Q830: BYTE;
	Q831: BYTE;
	Q832: BYTE;
	Q833: BYTE;
	Q834: BYTE;
	Q835: BYTE;
	Q836: BYTE;
	Q837: BYTE;
	Q838: BYTE;
	Q839: BYTE;
	Q840: BYTE;
	Q841: BYTE;
	Q842: BYTE;
	Q843: BYTE;
	Q844: BYTE;
	Q845: BYTE;
	Q846: BYTE;
	Q847: BYTE;
	Q848: BYTE;
	Q849: BYTE;
	Q850: BYTE;
	Q851: BYTE;
	Q852: BYTE;
	Q853: BYTE;
	Q854: BYTE;
	Q855: BYTE;
	Q856: BYTE;
	Q857: BYTE;
	Q858: BYTE;
	Q859: BYTE;
	Q860: BYTE;
	Q861: BYTE;
	Q862: BYTE;
	Q863: BYTE;
	Q864: BYTE;
	Q865: BYTE;
	Q866: BYTE;
	Q867: BYTE;
	Q868: BYTE;
	Q869: BYTE;
	Q870: BYTE;
	Q871: BYTE;
	Q872: BYTE;
	Q873: BYTE;
	Q874: BYTE;
	Q875: BYTE;
	Q876: BYTE;
	Q877: BYTE;
	Q878: BYTE;
	Q879: BYTE;
	Q880: BYTE;
	Q881: BYTE;
	Q882: BYTE;
	Q883: BYTE;
	Q884: BYTE;
	Q885: BYTE;
	Q886: BYTE;
	Q887: BYTE;
	Q888: BYTE;
	Q889: BYTE;
	Q890: BYTE;
	Q891: BYTE;
	Q892: BYTE;
	Q893: BYTE;
	Q894: BYTE;
	Q895: BYTE;
	Q896: BYTE;
	Q897: BYTE;
	Q898: BYTE;
	Q899: BYTE;
	Q900: BYTE;
	Q901: BYTE;
	Q902: BYTE;
	Q903: BYTE;
	Q904: BYTE;
	Q905: BYTE;
	Q906: BYTE;
	Q907: BYTE;
	Q908: BYTE;
	Q909: BYTE;
	Q910: BYTE;
	Q911: BYTE;
	Q912: BYTE;
	Q913: BYTE;
	Q914: BYTE;
	Q915: BYTE;
	Q916: BYTE;
	Q917: BYTE;
	Q918: BYTE;
	Q919: BYTE;
	Q920: BYTE;
	Q921: BYTE;
	Q922: BYTE;
	Q923: BYTE;
	Q924: BYTE;
	Q925: BYTE;
	Q926: BYTE;
	Q927: BYTE;
	Q928: BYTE;
	Q929: BYTE;
	Q930: BYTE;
	Q931: BYTE;
	Q932: BYTE;
	Q933: BYTE;
	Q934: BYTE;
	Q935: BYTE;
	Q936: BYTE;
	Q937: BYTE;
	Q938: BYTE;
	Q939: BYTE;
	Q940: BYTE;
	Q941: BYTE;
	Q942: BYTE;
	Q943: BYTE;
	Q944: BYTE;
	Q945: BYTE;
	Q946: BYTE;
	Q947: BYTE;
	Q948: BYTE;
	Q949: BYTE;
	Q950: BYTE;
	Q951: BYTE;
	Q952: BYTE;
	Q953: BYTE;
	Q954: BYTE;
	Q955: BYTE;
	Q956: BYTE;
	Q957: BYTE;
	Q958: BYTE;
	Q959: BYTE;
	Q960: BYTE;
	Q961: BYTE;
	Q962: BYTE;
	Q963: BYTE;
	Q964: BYTE;
	Q965: BYTE;
	Q966: BYTE;
	Q967: BYTE;
	Q968: BYTE;
	Q969: BYTE;
	Q970: BYTE;
	Q971: BYTE;
	Q972: BYTE;
	Q973: BYTE;
	Q974: BYTE;
	Q975: BYTE;
	Q976: BYTE;
	Q977: BYTE;
	Q978: BYTE;
	Q979: BYTE;
	Q980: BYTE;
	Q981: BYTE;
	Q982: BYTE;
	Q983: BYTE;
	Q984: BYTE;
	Q985: BYTE;
	Q986: BYTE;
	Q987: BYTE;
	Q988: BYTE;
	Q989: BYTE;
	Q990: BYTE;
	Q991: BYTE;
	Q992: BYTE;
	Q993: BYTE;
	Q994: BYTE;
	Q995: BYTE;
	Q996: BYTE;
	Q997: BYTE;
	Q998: BYTE;
	Q999: BYTE;
	Q1000: BYTE;
	Q1001: BYTE;
	Q1002: BYTE;
	Q1003: BYTE;
	Q1004: BYTE;
	Q1005: BYTE;
	Q1006: BYTE;
	Q1007: BYTE;
	Q1008: BYTE;
	Q1009: BYTE;
	Q1010: BYTE;
	Q1011: BYTE;
	Q1012: BYTE;
	Q1013: BYTE;
	Q1014: BYTE;
	Q1015: BYTE;
	Q1016: BYTE;
	Q1017: BYTE;
	Q1018: BYTE;
	Q1019: BYTE;
	Q1020: BYTE;
	Q1021: BYTE;
	Q1022: BYTE;
	Q1023: BYTE;
END_STRUCT
END_TYPE

// ---- Sil/PLC/GVL_PLC.TcGVL
{attribute 'linkalways'}
{attribute 'qualified_only'}
{attribute 'subsequent'}
{attribute 'pack_mode' := '1'}
VAR_GLOBAL
	Inputs : ST_PLCInputs;
	Outputs : ST_PLCOutputs;
END_VAR

// ---- FG_01/FG_01.TcPOU
FUNCTION_BLOCK FG_01

{region generated code}
VAR_INPUT
	B_SafetyGate1 : FB_SensorBinary;
	B_SafetyGate2 : FB_SensorBinary;
	P_Camera : FB_Camera;
	Y_Gate1 : FB_Cylinder;
	Y_Gate2 : FB_Cylinder;
	Y_Gripper : FB_Cylinder;
	Y_LaserMark : FB_DeviceByte;
	Y_Platform : FB_Cylinder;
	Y_ReaderWindow : FB_Cylinder;
END_VAR
{endregion}

{region generated code}
	InitRun();
	B_SafetyGate1();
	B_SafetyGate2();
	P_Camera();
	Y_Gate1();
	Y_Gate2();
	Y_Gripper();
	Y_LaserMark();
	Y_Platform();
	Y_ReaderWindow();
{endregion}

Mapping();

METHOD InitRun
{region generated code}
VAR_INST
	bInitRun : BOOL := TRUE;
END_VAR
{endregion}
{region generated code}
	IF NOT bInitRun THEN RETURN; END_IF
	bInitRun := FALSE;
{endregion}
END_METHOD

ACTION Mapping:
// ============================================================================
// FG_01 twin <-> PLCSIM Advanced process image.
//
// Addresses are the Siemens PLC tag tables in Siemens/_data/:
//   PLCTags_FG01.xlsx          the station's own cylinders
//   PLCTags_FG_Transport.xlsx  the two gates - see below
//
// GVL_PLC.Inputs / .Outputs are the PLC's process image seen from the twin side,
// so direction is baked into which side of the assignment the GVL sits on:
//   twin status -> GVL_PLC.Inputs    the PLC reads it
//   GVL_PLC.Outputs -> twin control  the PLC drives it
//
// THE GATES ARE MAPPED HERE, NOT IN FG_Transport. Y_Gate1 and Y_Gate2 moved into
// FG_01 with the twin and are members of THIS function block; the Siemens tag
// table still files their addresses under FG_TS_Gate_*, because a tag table is
// named for the PLC unit that owns the address, not for the twin group that owns
// the device. FG_Transport's Mapping used to assign them and could not compile.
// ============================================================================

// --- Y_Gripper - double solenoid, both coils and both limits ----------------
// InHome %I101.0 "geoeffnet" -> retracted = OPEN. WorkPos %Q101.1 "schliessen".
//
// THE RETRACT COIL IS NEW. The table gained HomePos %Q101.0 in this revision; it
// was missing before and the twin cylinder could never leave the extended limit
// once bExtend dropped, because a de-energised double solenoid does not spring
// back. Same fault, same fix, as the Beckhoff side.
GVL_PLC.Inputs.I101.0	:= Y_Gripper.bRetracted;
GVL_PLC.Inputs.I101.1	:= Y_Gripper.bExtended;
Y_Gripper.bRetract	:= GVL_PLC.Outputs.Q101.0;
Y_Gripper.bExtend	:= GVL_PLC.Outputs.Q101.1;

// --- Y_Platform - double solenoid, both coils and both limits ---------------
// InHome %I102.0 "hinten", InWork %I102.1 "vorne".
GVL_PLC.Inputs.I102.0	:= Y_Platform.bRetracted;
GVL_PLC.Inputs.I102.1	:= Y_Platform.bExtended;
Y_Platform.bRetract	:= GVL_PLC.Outputs.Q102.0;
Y_Platform.bExtend	:= GVL_PLC.Outputs.Q102.1;

// --- Y_ReaderWindow - double solenoid, both coils, ONE limit ----------------
// WorkPos %Q103.1 "Position zum Code Lesen". HomePos %Q103.0 is new in this
// revision, for the same reason as Y_Gripper's above.
//
// THE TABLE HAS NO Y_ReaderWindow_InHome. bRetracted is therefore not published
// and the control PLC cannot see the window fully back - only that it is not at
// the read position. Add %I103.0 to PLCTags_FG01.xlsx to close that.
GVL_PLC.Inputs.I103.1	:= Y_ReaderWindow.bExtended;
Y_ReaderWindow.bRetract	:= GVL_PLC.Outputs.Q103.0;
Y_ReaderWindow.bExtend	:= GVL_PLC.Outputs.Q103.1;

// --- Y_Gate1 / Y_Gate2 - single solenoid, spring return ---------------------
// EXTEND CLOSES the gate and the spring opens it, so the coil is the CLOSING
// command and both limits are read:
//   InHome %I100x.0 "geoeffnet"  -> retracted = open
//   InWork %I100x.1 "geschlossen" -> extended  = closed
//   WorkPos %Q100x.1 "Schliessen" -> the close coil
//
// THE COIL IS %Q100x.1, NOT %Q100x.0. The previous mapping drove bit 0, which is
// not a tag in the table at all, so the gates never closed.
Y_Gate1.bExtend	:= GVL_PLC.Outputs.Q1001.1;
GVL_PLC.Inputs.I1001.0	:= Y_Gate1.bRetracted;
GVL_PLC.Inputs.I1001.1	:= Y_Gate1.bExtended;

Y_Gate2.bExtend	:= GVL_PLC.Outputs.Q1002.1;
GVL_PLC.Inputs.I1002.0	:= Y_Gate2.bRetracted;
GVL_PLC.Inputs.I1002.1	:= Y_Gate2.bExtended;

// --- P_Camera - the identify read -------------------------------------------
// What the part must be carrying. FG_01 is the identify station: the twin's
// DataReader reads the payload's SerialNumber key, and Assembly Part 1 carries
// 60. A pallet with no part, or a part with no serial number, reads 0 and fails.
//
// SET HERE AND NOT IN InitRun BECAUSE Mapping IS THE ONLY ACTION WE OWN - OC
// Assistant regenerates everything inside the {region generated code} blocks on
// the next twin regeneration.
P_Camera.nExpectedData := 60;

// TODO: NO ADDRESS IN PLCTags_FG01.xlsx for P_Camera (FB_Camera).
// Four bits are needed and the bit roles are fixed by FB_AbstractCamera:
//   OUT bit 0 Enable   bit 1 Trigger
//   IN  bit 0 Ready    bit 1 Busy   bit 2 ResultValid   bit 3 ResultOK
// Add one input byte and one output byte to the table, then:
//   P_Camera.bEnable  := GVL_PLC.Outputs.Q<n>.0;
//   P_Camera.bTrigger := GVL_PLC.Outputs.Q<n>.1;
//   GVL_PLC.Inputs.I<n>.0 := P_Camera.bReady;
//   GVL_PLC.Inputs.I<n>.1 := P_Camera.bBusy;
//   GVL_PLC.Inputs.I<n>.2 := P_Camera.bResultValid;
//   GVL_PLC.Inputs.I<n>.3 := P_Camera.bResultOK;
// Until then the station cannot read a part and FG_01 cannot run.

// TODO: NO ADDRESS IN PLCTags_FG01.xlsx for Y_LaserMark (FB_DeviceByte).
// One control byte out, one status byte back; only control bit 0 is used - held
// high for 1 s it applies the mark - and there are NO status bits, so the PLC
// gets no confirmation that the laser fired. Needs one output byte:
//   Y_LaserMark.nControlData.0 := GVL_PLC.Outputs.Q<n>.0;

// TODO: NO ADDRESS IN PLCTags_FG01.xlsx for B_SafetyGate1 / B_SafetyGate2
// (FB_SensorBinary). These are the independent gate-position monitors the laser
// interlock reads; without them the interlock has only the cylinder limits,
// which is exactly the single-source-of-truth the second sensor exists to avoid.
//   GVL_PLC.Inputs.I<n>.<b> := B_SafetyGate1.bValue;
//   GVL_PLC.Inputs.I<n>.<b> := B_SafetyGate2.bValue;
END_ACTION

END_FUNCTION_BLOCK

// ---- Library/FB_Camera.TcPOU
// ============================================================================
// Inspection camera - the TWIN side of the vision-sensor interface.
//
// It sits between two interfaces that are NOT the same shape, and translating
// between them is its entire job.
//
// Below it, the Unity DataReader (Preliy.Demo.DataReader). Two bits down, two
// bits and a 64 bit datum back - an echo and a value, nothing more:
//
//   Control 0  Enable            Status 0  Enabled     (echo of Enable)
//   Control 1  Trigger           Status 1  Triggered   (echo of Trigger)
//                                StatusData  the payload datum read for _key,
//                                            0 when there is no payload, no
//                                            such key, or the trigger is low
//
// Above it, FB_AbstractCamera in OC_PLC, which expects a real handshake:
//
//   Output 0  Enable             Input 0  Ready
//   Output 1  Trigger            Input 1  Busy
//                                Input 2  ResultValid
//                                Input 3  ResultOK
//
// THE TWIN DOES NOT KNOW ABOUT READY, BUSY OR A VERDICT. The DataReader only
// echoes what it was asked and hands over a number. Ready, Busy, ResultValid and
// ResultOK are synthesised here, out of that echo plus one exposure timer plus
// the comparison against nExpectedData. That is the point of this block: the twin
// stays a dumb sensor and the emulated device carries the protocol.
//
// bResultValid USED TO BE THE CONSTANT TRUE, which meant the control PLC could
// never tell "no verdict yet" from "verdict says no" - the exact distinction
// FG_02's three fault codes are built on. It is now a real latch: it goes up when
// the exposure completes, holds while the trigger is held, and drops when the
// trigger is released.
//
// Bit assignment on the wire is decided in the calling group's Mapping action.
// Both halves have to agree on it; nothing checks it for you.
// ============================================================================
FUNCTION_BLOCK FB_Camera EXTENDS FB_LinkDataLWord
VAR_INPUT
	// Commanded state, from the control PLC via the group Mapping action.
	bEnable			: BOOL;
	bTrigger		: BOOL;
	// The datum the part must carry for this shot to pass. Compared as a signed
	// integer against StatusData, which Unity writes as a C# long.
	//
	// A VALUE OF 0 MAKES THE VERDICT MEANINGLESS: an absent payload, a key the
	// payload does not carry and a failed parse all read back 0, so a part that
	// was never inspected would report OK. Configure a real value in Mapping.
	nExpectedData	: LINT;
	// How long the shot takes. Modelled, not measured - a vision sensor of this
	// class answers in the low hundreds of ms. It must stay well inside FG_02's
	// 3 s shot budget, and it must be non-zero, or Busy would never be observable
	// and the control side could not distinguish a shot from a stuck trigger.
	tExposure		: TIME := T#2000MS;
END_VAR
VAR_OUTPUT
	// The twin's own echo, straight off the status byte.
	bEnabled		: BOOL;
	bTriggered		: BOOL;
	// The synthesised handshake. These are what the group maps to the terminal.
	bReady			: BOOL;
	bBusy			: BOOL;
	bResultValid	: BOOL;
	bResultOK		: BOOL;
	// The datum latched by the last completed shot, held for as long as the
	// verdict is. Not on the wire - the interface is four bits - but it is what
	// makes a NOK diagnosable when watching the SIM online.
	nResult			: LINT;
END_VAR
VAR
	ExposureTimer	: TON;
END_VAR

// --- command down to the twin -----------------------------------------------
Control.0 := bEnable;
Control.1 := bTrigger;

// --- the twin's answer, unmodified ------------------------------------------
bEnabled	:= Status.0;
bTriggered	:= Status.1;

// --- the shot ----------------------------------------------------------------
// The timer is armed on the COMMAND and the ECHO together. Both matter:
//
//   bEnable / bTrigger  - dropping the trigger has to reset the exposure on the
//                         same scan. Arming on bTriggered alone would leave the
//                         timer running through the scans the twin takes to
//                         echo the release, and an already-elapsed TON re-latches
//                         a stale verdict the moment it is looked at again.
//   bEnabled/bTriggered - the twin has to have actually accepted the command. If
//                         Unity is not connected the status byte stays 0, no
//                         exposure ever starts, Ready never comes and FG_02
//                         raises fault 2. That is the honest outcome.
//
// NOT bResultValid stops the timer once a verdict is out, so the verdict is
// latched once and then stands still rather than being recomputed every scan.
ExposureTimer(
	IN	:= bEnable AND bTrigger AND bEnabled AND bTriggered AND NOT bResultValid,
	PT	:= tExposure);

IF ExposureTimer.Q THEN
	// StatusData is a bit string on this side and a signed long on Unity's.
	// Convert rather than compare across types - LWORD against LINT is not a
	// comparison the compiler will do for you.
	nResult			:= LWORD_TO_LINT(StatusData);
	bResultOK		:= nResult = nExpectedData;
	bResultValid	:= TRUE;
END_IF

// The verdict is released by the trigger being released - which is also what
// tells the twin to clear its value - or by the camera being powered down.
IF NOT bTrigger OR NOT bEnable THEN
	bResultValid	:= FALSE;
	bResultOK		:= FALSE;
	nResult			:= 0;
END_IF

// --- the handshake bits -------------------------------------------------------
// Both are DERIVED EVERY SCAN, never remembered. A stored flag maintained in one
// branch is stale in every other one.
//
// Ready is permission to trigger: powered, idle, and holding no unread verdict.
// Busy is the exposure in progress: triggered and no verdict out yet.
bBusy	:= bEnable AND bEnabled AND bTriggered AND NOT bResultValid;
bReady	:= bEnable AND bEnabled AND NOT bTriggered AND NOT bResultValid;

END_FUNCTION_BLOCK

// ---- FG_02/FG_02.TcPOU
FUNCTION_BLOCK FG_02

{region generated code}
VAR_INPUT
	P_Camera : FB_Camera;
END_VAR
{endregion}

{region generated code}
	InitRun();
	P_Camera();
{endregion}

Mapping();

METHOD InitRun
{region generated code}
VAR_INST
	bInitRun : BOOL := TRUE;
END_VAR
{endregion}
{region generated code}
	IF NOT bInitRun THEN RETURN; END_IF
	bInitRun := FALSE;
{endregion}
END_METHOD

ACTION Mapping:
// ============================================================================
// FG_02 twin <-> PLCSIM Advanced process image.
//
// One device, and it has no address yet. There is NO PLCTags_FG02.xlsx in
// Siemens/_data/ at all - FG_02 is the only group with no tag table.
// ============================================================================

// --- P_Camera - the mark verification read ----------------------------------
// FG_02 inspects the mark FG_01 applied: the laser writes LaserMark := 240 onto
// the payload, this station reads that key back and passes only on 240. A part
// that skipped FG_01, or whose mark failed, reads 0 and is a NOK.
//
// SET HERE AND NOT IN InitRun BECAUSE Mapping IS THE ONLY ACTION WE OWN - OC
// Assistant regenerates everything inside the {region generated code} blocks on
// the next twin regeneration.
P_Camera.nExpectedData := 240;

// TODO: NO TAG TABLE FOR FG_02. Add PLCTags_FG02.xlsx with one input byte and
// one output byte, then wire the four bits. The bit roles are fixed by
// FB_AbstractCamera and are IDENTICAL in FG_01, FG_02 and FG_05:
//   OUT bit 0 Enable   bit 1 Trigger
//   IN  bit 0 Ready    bit 1 Busy   bit 2 ResultValid   bit 3 ResultOK
//
//   P_Camera.bEnable  := GVL_PLC.Outputs.Q<n>.0;
//   P_Camera.bTrigger := GVL_PLC.Outputs.Q<n>.1;
//   GVL_PLC.Inputs.I<n>.0 := P_Camera.bReady;
//   GVL_PLC.Inputs.I<n>.1 := P_Camera.bBusy;
//   GVL_PLC.Inputs.I<n>.2 := P_Camera.bResultValid;
//   GVL_PLC.Inputs.I<n>.3 := P_Camera.bResultOK;
END_ACTION

END_FUNCTION_BLOCK

// ---- FG_03/FG_03.TcPOU
FUNCTION_BLOCK FG_03

{region generated code}
VAR_INPUT
	B_Detect1 : FB_SensorBinary;
	B_Detect2 : FB_SensorBinary;
	Y_AxisR1 : FB_Cylinder;
	Y_AxisX1 : FB_Cylinder;
	Y_AxisX2 : FB_Cylinder;
	Y_AxisY1 : FB_Cylinder;
	Y_AxisY2 : FB_Cylinder;
	Y_Gripper1 : FB_Cylinder;
	Y_Gripper2 : FB_Cylinder;
END_VAR
{endregion}

{region generated code}
	InitRun();
	B_Detect1();
	B_Detect2();
	Y_AxisR1();
	Y_AxisX1();
	Y_AxisX2();
	Y_AxisY1();
	Y_AxisY2();
	Y_Gripper1();
	Y_Gripper2();
{endregion}

Mapping();

METHOD InitRun
{region generated code}
VAR_INST
	bInitRun : BOOL := TRUE;
END_VAR
{endregion}
{region generated code}
	IF NOT bInitRun THEN RETURN; END_IF
	bInitRun := FALSE;
{endregion}
END_METHOD

ACTION Mapping:
// ============================================================================
// FG_03 twin <-> PLCSIM Advanced process image.
//
// Addresses: Siemens/_data/PLCTags_FG03.xlsx. The only group whose cylinders are
// COMPLETE in the table - all seven have both limits and both coils:
//   InHome  %I3xx.0 -> bRetracted      HomePos %Q3xx.0 -> bRetract
//   InWork  %I3xx.1 -> bExtended       WorkPos %Q3xx.1 -> bExtend
//
// THE AXIS NAMES ARE A TRAP. Arm 1 is X1/Y1/R1 and arm 2 is X2/Y2, but R1 is the
// ROTATION shared by the transfer, not "arm 1's rotation". Read
// _docs/reference/fg-03-behaviour.md before writing control code against these.
// ============================================================================

// --- Y_AxisR1 - double solenoid ---------------------------------------------
GVL_PLC.Inputs.I301.0	:= Y_AxisR1.bRetracted;
GVL_PLC.Inputs.I301.1	:= Y_AxisR1.bExtended;
Y_AxisR1.bRetract	:= GVL_PLC.Outputs.Q301.0;
Y_AxisR1.bExtend	:= GVL_PLC.Outputs.Q301.1;

// --- Y_AxisX1 - double solenoid ---------------------------------------------
GVL_PLC.Inputs.I302.0	:= Y_AxisX1.bRetracted;
GVL_PLC.Inputs.I302.1	:= Y_AxisX1.bExtended;
Y_AxisX1.bRetract	:= GVL_PLC.Outputs.Q302.0;
Y_AxisX1.bExtend	:= GVL_PLC.Outputs.Q302.1;

// --- Y_AxisY1 - double solenoid ---------------------------------------------
GVL_PLC.Inputs.I303.0	:= Y_AxisY1.bRetracted;
GVL_PLC.Inputs.I303.1	:= Y_AxisY1.bExtended;
Y_AxisY1.bRetract	:= GVL_PLC.Outputs.Q303.0;
Y_AxisY1.bExtend	:= GVL_PLC.Outputs.Q303.1;

// --- Y_AxisX2 - double solenoid ---------------------------------------------
GVL_PLC.Inputs.I304.0	:= Y_AxisX2.bRetracted;
GVL_PLC.Inputs.I304.1	:= Y_AxisX2.bExtended;
Y_AxisX2.bRetract	:= GVL_PLC.Outputs.Q304.0;
Y_AxisX2.bExtend	:= GVL_PLC.Outputs.Q304.1;

// --- Y_AxisY2 - double solenoid ---------------------------------------------
GVL_PLC.Inputs.I305.0	:= Y_AxisY2.bRetracted;
GVL_PLC.Inputs.I305.1	:= Y_AxisY2.bExtended;
Y_AxisY2.bRetract	:= GVL_PLC.Outputs.Q305.0;
Y_AxisY2.bExtend	:= GVL_PLC.Outputs.Q305.1;

// --- Y_Gripper1 - double solenoid, the PLACING arm --------------------------
// The jaws reach .bExtended closed on NOTHING sooner than closed on a part, so
// this limit is not a grip witness. Only B_Detect1 says a part is held.
GVL_PLC.Inputs.I306.0	:= Y_Gripper1.bRetracted;
GVL_PLC.Inputs.I306.1	:= Y_Gripper1.bExtended;
Y_Gripper1.bRetract	:= GVL_PLC.Outputs.Q306.0;
Y_Gripper1.bExtend	:= GVL_PLC.Outputs.Q306.1;

// --- Y_Gripper2 - double solenoid -------------------------------------------
GVL_PLC.Inputs.I307.0	:= Y_Gripper2.bRetracted;
GVL_PLC.Inputs.I307.1	:= Y_Gripper2.bExtended;
Y_Gripper2.bRetract	:= GVL_PLC.Outputs.Q307.0;
Y_Gripper2.bExtend	:= GVL_PLC.Outputs.Q307.1;

// TODO: NO ADDRESS IN PLCTags_FG03.xlsx for B_Detect1 / B_Detect2
// (FB_SensorBinary). THESE ARE THE GRIP WITNESSES and their absence is the
// worst gap in this table: a gripper cylinder reaching .Extended proves nothing
// about whether a part is held, and FG_03's reset branches on exactly these two
// bits at Resetting step 0. Without them the station cannot reset safely with a
// part in a gripper. See _docs/reference/gripper-station-reset.md.
//   GVL_PLC.Inputs.I<n>.<b> := B_Detect1.bValue;
//   GVL_PLC.Inputs.I<n>.<b> := B_Detect2.bValue;
END_ACTION

END_FUNCTION_BLOCK

// ---- FG_04/FG_04.TcPOU
FUNCTION_BLOCK FG_04
{region generated code}
VAR_INPUT
	B_NIO : FB_SensorBinary;
	Y_AxisZ : FB_Cylinder;
END_VAR
{endregion}

{region generated code}
	InitRun();
	B_NIO();
	Y_AxisZ();
{endregion}

Mapping();

METHOD InitRun
{region generated code}
VAR_INST
	bInitRun : BOOL := TRUE;
END_VAR
{endregion}
{region generated code}
	IF NOT bInitRun THEN RETURN; END_IF
	bInitRun := FALSE;
{endregion}
END_METHOD

ACTION Mapping:
// ============================================================================
// FG_04 twin <-> PLCSIM Advanced process image.
//
// Addresses: Siemens/_data/PLCTags_FG04.xlsx.
//
// The press and its verdict. Y_AxisZ is a double solenoid so that an abort
// mid-stroke leaves it where it is instead of letting a spring drive it further
// into the part - which is why the retract coil below has to be driven and not
// left to a spring that does not exist.
// ============================================================================

// --- Y_AxisZ - double solenoid, both coils and both limits ------------------
// InHome %I401.0 and HomePos %Q401.0 are BOTH NEW in this revision of the table.
// Before them the press had no way back: it reported only the bottom limit and
// the retract coil did not exist, so once bExtend dropped the twin cylinder held
// its extended position for ever.
GVL_PLC.Inputs.I401.0	:= Y_AxisZ.bRetracted;
GVL_PLC.Inputs.I401.1	:= Y_AxisZ.bExtended;
Y_AxisZ.bRetract	:= GVL_PLC.Outputs.Q401.0;
Y_AxisZ.bExtend	:= GVL_PLC.Outputs.Q401.1;

// TODO: NO ADDRESS IN PLCTags_FG04.xlsx for B_NIO (FB_SensorBinary).
// B_NIO IS NOT A SENSOR READING, it is a VERDICT: the twin's seating sensor is
// not a PLC symbol at all - it feeds PartPressDetector inside Unity, which
// publishes the conclusion here as one bit. Active means the press bottomed with
// nothing correctly seated, and it is only meaningful at the bottom limit with
// the hold expired. Without it FG_04 presses and never judges.
//   GVL_PLC.Inputs.I<n>.<b> := B_NIO.bValue;
END_ACTION

END_FUNCTION_BLOCK

// ---- FG_05/FG_05.TcPOU
FUNCTION_BLOCK FG_05

{region generated code}
VAR_INPUT
	B_Detect : FB_SensorBinary;
	B_Part : FB_SensorBinary;
	P_Camera : FB_Camera;
	Y_AxisR : FB_Cylinder;
	Y_AxisX : FB_Cylinder;
	Y_AxisZ1 : FB_Cylinder;
	Y_AxisZ2 : FB_Cylinder;
	Y_CapsSource : FB_DeviceByte;
	Y_CapsSourceStopper : FB_Cylinder;
	Y_Gripper : FB_Cylinder;
END_VAR
{endregion}

{region generated code}
	InitRun();
	B_Detect();
	B_Part();
	P_Camera();
	Y_AxisR();
	Y_AxisX();
	Y_AxisZ1();
	Y_AxisZ2();
	Y_CapsSource();
	Y_CapsSourceStopper();
	Y_Gripper();
{endregion}

Mapping();

METHOD InitRun
{region generated code}
VAR_INST
	bInitRun : BOOL := TRUE;
END_VAR
{endregion}
{region generated code}
	IF NOT bInitRun THEN RETURN; END_IF
	bInitRun := FALSE;
{endregion}
END_METHOD

ACTION Mapping:
// ============================================================================
// FG_05 twin <-> PLCSIM Advanced process image.
//
// Addresses: Siemens/_data/PLCTags_FG05.xlsx.
//
// Capping. Four double solenoids on the handler, a single-acting stopper on the
// cap feed, and the bunker - which is an FB_DeviceByte, not a drive, and gained
// its two control bits in this revision of the table.
// ============================================================================

// --- B_Part - cap present at the pick position, on the FEED -----------------
// NOT the same question as B_Detect below and not interchangeable with it:
// B_Part is on the feed and reports the NEXT cap as soon as this one is lifted
// away.
GVL_PLC.Inputs.I500.0	:= B_Part.bValue;

// --- Y_AxisR - double solenoid ----------------------------------------------
GVL_PLC.Inputs.I501.0	:= Y_AxisR.bRetracted;
GVL_PLC.Inputs.I501.1	:= Y_AxisR.bExtended;
Y_AxisR.bRetract	:= GVL_PLC.Outputs.Q501.0;
Y_AxisR.bExtend	:= GVL_PLC.Outputs.Q501.1;

// --- Y_AxisX - double solenoid ----------------------------------------------
GVL_PLC.Inputs.I502.0	:= Y_AxisX.bRetracted;
GVL_PLC.Inputs.I502.1	:= Y_AxisX.bExtended;
Y_AxisX.bRetract	:= GVL_PLC.Outputs.Q502.0;
Y_AxisX.bExtend	:= GVL_PLC.Outputs.Q502.1;

// --- Y_AxisZ1 - double solenoid ---------------------------------------------
GVL_PLC.Inputs.I503.0	:= Y_AxisZ1.bRetracted;
GVL_PLC.Inputs.I503.1	:= Y_AxisZ1.bExtended;
Y_AxisZ1.bRetract	:= GVL_PLC.Outputs.Q503.0;
Y_AxisZ1.bExtend	:= GVL_PLC.Outputs.Q503.1;

// --- Y_AxisZ2 - double solenoid ---------------------------------------------
GVL_PLC.Inputs.I504.0	:= Y_AxisZ2.bRetracted;
GVL_PLC.Inputs.I504.1	:= Y_AxisZ2.bExtended;
Y_AxisZ2.bRetract	:= GVL_PLC.Outputs.Q504.0;
Y_AxisZ2.bExtend	:= GVL_PLC.Outputs.Q504.1;

// --- Y_CapsSourceStopper - both coils, ONE limit ----------------------------
//   InHome  %I505.0 "GS = Kaps koennen vereinzelt werden"
//   HomePos %Q505.0 - NEW in this revision, the missing return coil
//   WorkPos %Q505.1 "AS = Vereinzelung kann geleert werden"
//
// THE TABLE HAS NO Y_CapsSourceStopper_InWork, so bExtended is not published and
// the control PLC cannot see the stopper fully open - only that it has left the
// singulating position. Add %I505.1 to close that.
GVL_PLC.Inputs.I505.0	:= Y_CapsSourceStopper.bRetracted;
Y_CapsSourceStopper.bRetract	:= GVL_PLC.Outputs.Q505.0;
Y_CapsSourceStopper.bExtend	:= GVL_PLC.Outputs.Q505.1;

// --- Y_Gripper - double solenoid --------------------------------------------
// .bExtended is jaws closed, on a cap or on nothing. Only B_Detect witnesses a
// held cap, and B_Detect has no address - see the TODO at the bottom.
GVL_PLC.Inputs.I506.0	:= Y_Gripper.bRetracted;
GVL_PLC.Inputs.I506.1	:= Y_Gripper.bExtended;
Y_Gripper.bRetract	:= GVL_PLC.Outputs.Q506.0;
Y_Gripper.bExtend	:= GVL_PLC.Outputs.Q506.1;

// --- Y_CapsSource - the bunker, FB_DeviceByte -------------------------------
// NEW IN THIS REVISION: M_Bunker %Q507.0 and M_Conveyor %Q507.1. This device is
// an FB_DeviceByte, so the PLC drives BITS OF ITS CONTROL BYTE, not two separate
// coils - the twin's authored BitLayout fixes which bit is which:
//   bit 0  the vibration table that feeds the bunker   ("Sortiertopf ein")
//   bit 1  the short caps conveyor to the pick position ("Linearfoerderer ein")
//
// The bunker reports NOTHING back - there are no status bits and no tags for
// any, which is correct rather than missing. It runs continuously while enabled;
// it is not started per cap.
Y_CapsSource.nControlData.0	:= GVL_PLC.Outputs.Q507.0;
Y_CapsSource.nControlData.1	:= GVL_PLC.Outputs.Q507.1;

// --- P_Camera - the assembly identification read ----------------------------
// IT READS THE ASSEMBLY ON THE PALLET, NOT THE CAP. The camera is mounted on the
// feed side but looks across at the pallet, and the key it reads - CapsID - is
// authored on Assembly Part 1, which carries 810. So the read answers "which cap
// does this assembly want", and the station passes only on the type it is set up
// to fit. An empty pallet reads 0 and fails.
//
// SET HERE AND NOT IN InitRun BECAUSE Mapping IS THE ONLY ACTION WE OWN - OC
// Assistant regenerates everything inside the {region generated code} blocks on
// the next twin regeneration.
P_Camera.nExpectedData := 810;

// TODO: NO ADDRESS IN PLCTags_FG05.xlsx for P_Camera (FB_Camera).
// Bit roles are fixed by FB_AbstractCamera and identical in FG_01/02/05:
//   OUT bit 0 Enable   bit 1 Trigger
//   IN  bit 0 Ready    bit 1 Busy   bit 2 ResultValid   bit 3 ResultOK
//   P_Camera.bEnable  := GVL_PLC.Outputs.Q<n>.0;
//   P_Camera.bTrigger := GVL_PLC.Outputs.Q<n>.1;
//   GVL_PLC.Inputs.I<n>.0 := P_Camera.bReady;
//   GVL_PLC.Inputs.I<n>.1 := P_Camera.bBusy;
//   GVL_PLC.Inputs.I<n>.2 := P_Camera.bResultValid;
//   GVL_PLC.Inputs.I<n>.3 := P_Camera.bResultOK;
// The read comes FIRST in this station's cycle, so without it FG_05 cannot start.

// TODO: NO ADDRESS IN PLCTags_FG05.xlsx for B_Detect (FB_SensorBinary).
// Cap held in the gripper's JAWS - the grip witness. FG_05's reset branches on
// it at Resetting step 0, and the cylinder limit cannot answer the question.
//   GVL_PLC.Inputs.I<n>.<b> := B_Detect.bValue;
END_ACTION

END_FUNCTION_BLOCK

// ---- FG_System/FG_System.TcPOU
FUNCTION_BLOCK FG_System

{region generated code}
VAR_INPUT
	B_SafetyDoor11 : FB_Lock;
	B_SafetyDoor12 : FB_Lock;
	B_SafetyDoor13 : FB_Lock;
	B_SafetyDoor21 : FB_Lock;
	B_SafetyDoor22 : FB_Lock;
	B_SafetyDoor23 : FB_Lock;
	H_ControlPanel : FB_Panel;
	H_SignalTower : FB_Panel;
	SS_EStop1 : FB_Button;
	SS_EStop2 : FB_Button;
END_VAR
{endregion}

{region generated code}
	InitRun();
	B_SafetyDoor11();
	B_SafetyDoor12();
	B_SafetyDoor13();
	B_SafetyDoor21();
	B_SafetyDoor22();
	B_SafetyDoor23();
	H_ControlPanel();
	H_SignalTower();
	SS_EStop1();
	SS_EStop2();
{endregion}

Mapping();

METHOD InitRun
{region generated code}
VAR_INST
	bInitRun : BOOL := TRUE;
END_VAR
{endregion}
{region generated code}
	IF NOT bInitRun THEN RETURN; END_IF
	bInitRun := FALSE;
{endregion}
END_METHOD

ACTION Mapping:
// ============================================================================
// FG_System twin <-> PLCSIM Advanced process image.
//
// Addresses: Siemens/_data/PLCTags_ControlPanel.xlsx.
//
// THIS IS THE SIEMENS PANEL, NOT THE BECKHOFF ONE. The two scenes differ in
// exactly one node: H_ControlPanel here resolves to
// MAIN.FG_System.H_ControlPanel_Siemens, a PanelSampler over SEVEN controls, of
// which one - OP MODE - is a SwitchRotary and not a button. The Beckhoff panel is
// eight PackML buttons and its bit order is a different thing entirely; do not
// carry a bit layout across from it.
//
// Bit order below is the twin's own _components order, read from
// Unity/Assets/StreamingAssets/VC_Demo_1_Siemens_1_Context.json. It lines up
// one-for-one with BT1..BT7 in the tag table, which is why no lookup is needed:
//   bit 0 CONTROL ON/OFF   bit 1 OP MODE (rotary)   bit 2 SINGLE STEP
//   bit 3 AUTO START       bit 4 AUTO STOP          bit 5 ERROR ACK
//   bit 6 RESET
//
// Reordering that _components list changes the PLC bit assignment. Nothing here
// checks it for you.
// ============================================================================

// --- H_ControlPanel: the controls -> %I0.1 .. %I0.7 -------------------------
GVL_PLC.Inputs.I0.1	:= H_ControlPanel.nStatusData.0;	// BT1 CONTROL ON/OFF
GVL_PLC.Inputs.I0.2	:= H_ControlPanel.nStatusData.1;	// BT2 OP MODE  1=Auto / 0=Hand
GVL_PLC.Inputs.I0.3	:= H_ControlPanel.nStatusData.2;	// BT3 SINGLE STEP
GVL_PLC.Inputs.I0.4	:= H_ControlPanel.nStatusData.3;	// BT4 AUTO START
GVL_PLC.Inputs.I0.5	:= H_ControlPanel.nStatusData.4;	// BT5 AUTO STOP
GVL_PLC.Inputs.I0.6	:= H_ControlPanel.nStatusData.5;	// BT6 ERROR ACK
GVL_PLC.Inputs.I0.7	:= H_ControlPanel.nStatusData.6;	// BT7 RESET

// --- H_ControlPanel: the button lamps -> %Q0.1 .. %Q0.7 ---------------------
// Same bit order as the controls above, so bit n lights the control bit n reads.
// BIT 1 IS DELIBERATELY ABSENT: OP MODE is a rotary switch and has no lamp, and
// the tag table has no BT2 light either. That gap is correct, not missing.
H_ControlPanel.nControlData.0	:= GVL_PLC.Outputs.Q0.1;	// BT1 "Steuerung laeuft" (gruen)
H_ControlPanel.nControlData.2	:= GVL_PLC.Outputs.Q0.3;	// BT3 "Einzelschritt laeuft" (gruen)
H_ControlPanel.nControlData.3	:= GVL_PLC.Outputs.Q0.4;	// BT4 "Automatik laeuft" (gruen)
H_ControlPanel.nControlData.4	:= GVL_PLC.Outputs.Q0.5;	// BT5 "Automatik Stop laeuft" (blau)
H_ControlPanel.nControlData.5	:= GVL_PLC.Outputs.Q0.6;	// BT6 "Lampe Stoerung" (rot)
H_ControlPanel.nControlData.6	:= GVL_PLC.Outputs.Q0.7;	// BT7 "Grundstellungsfahrt laeuft" (gruen)

// --- H_SignalTower -> %Q1.1 .. %Q1.3 ----------------------------------------
// ALL THREE OF THESE ASSIGNMENTS WERE WRONG and are corrected here. The tower is
// FOUR lamps and its bit order, verified 2026-08-20 against the live
// PanelSampler._components list and identical in both vendor scenes, is:
//   bit 0 RED   bit 1 YELLOW   bit 2 BLUE   bit 3 GREEN
//
// The previous mapping assumed three lamps with GREEN at bit 2 - the twin's own
// authored prose said so until it was corrected - and then drove bit 2 from
// %Q1.0, which is not a tower tag at all but BT8's own button lamp. So RED lit
// on the yellow tag, YELLOW on the green tag, and the immediate-stop button lamp
// lit the tower.
H_SignalTower.nControlData.0	:= GVL_PLC.Outputs.Q1.3;	// RED    "Stoerung"
H_SignalTower.nControlData.1	:= GVL_PLC.Outputs.Q1.2;	// YELLOW "Einrichten aktiv"
H_SignalTower.nControlData.3	:= GVL_PLC.Outputs.Q1.1;	// GREEN  "Automatik laeuft"

// BLUE is bit 2 and has NO Siemens tag. The machine's indication contract uses it
// for Low Material / Material Exhausted - see _docs/reference/state-lamp.md - and
// FG_System exposes those inputs but never sets them, so an unmapped blue lamp
// loses nothing today. Add %Q1.4 if the material model ever becomes real.

// TODO: BT8_ImmediateStop %I1.0 / BT8_ImmediateStopLight %Q1.0 HAVE NO TWIN
// SOURCE. The Siemens panel is seven controls and BT8 is not one of them, so
// nothing in H_ControlPanel_Siemens can drive it. The only plausible candidates
// are SS_EStop1 / SS_EStop2, but they are two latching mushrooms and this is one
// bit on an illuminated PUSH button ("Sofort Halt"), which is a different device
// doing a different job. THIS IS A QUESTION FOR THE USER, not something to infer:
// either the panel needs an eighth control authored in the Unity scene, or BT8
// is a real E-stop channel and the two mushrooms have to be combined - and which
// one it is decides whether the cell can be stopped at all.

// TODO: NO ADDRESS IN PLCTags_ControlPanel.xlsx for SS_EStop1 / SS_EStop2
// (FB_Button). One input and one lamp coil each. On the Beckhoff side the twin
// value is INVERTED on the way in, so the PLC reads a real NC mushroom - TRUE
// while healthy, FALSE while latched - and FG_System sets Inverted := TRUE to
// match. Do the same here, and do not drop the NOT without clearing that too:
//   GVL_PLC.Inputs.I<n>.<b> := NOT SS_EStop1.bValue;
//   GVL_PLC.Inputs.I<n>.<b> := NOT SS_EStop2.bValue;
//   SS_EStop1.bEnable := GVL_PLC.Outputs.Q<n>.<b>;   // bEnable IS the lamp
//   SS_EStop2.bEnable := GVL_PLC.Outputs.Q<n>.<b>;

// TODO: NO ADDRESS IN PLCTags_ControlPanel.xlsx for the six B_SafetyDoor*
// (FB_Lock). Each needs TWO inputs and ONE output - closed, locked, and the lock
// coil - because secure means BOTH: closed alone does not make a guard secure.
// Twelve inputs and six outputs in twin order 11/12/13 then 21/22/23:
//   GVL_PLC.Inputs.I<n>.<b> := B_SafetyDoor11.bClosed;
//   GVL_PLC.Inputs.I<n>.<b> := B_SafetyDoor11.bLocked;
//   B_SafetyDoor11.bLock := GVL_PLC.Outputs.Q<n>.<b>;
//   ... and so on for 12, 13, 21, 22, 23.
// Until these exist the cell has no guard monitoring and no way to release a
// door for maintenance. See _docs/reference/fg-system-safety.md for who owns
// which half of that decision.
END_ACTION

END_FUNCTION_BLOCK

// ---- FG_Transport/FG_Transport.TcPOU
FUNCTION_BLOCK FG_Transport

{region generated code}
VAR_INPUT
	Index01_B_Detect : FB_SensorBinary;
	Index01_B_Exit : FB_SensorBinary;
	Index01_Y_Lift : FB_Cylinder;
	Index01_Y_Stopper : FB_Cylinder;
	Index02_B_Detect : FB_SensorBinary;
	Index02_B_Exit : FB_SensorBinary;
	Index02_Y_Lift : FB_Cylinder;
	Index02_Y_Stopper : FB_Cylinder;
	Index03_B_Detect : FB_SensorBinary;
	Index03_B_Exit : FB_SensorBinary;
	Index03_Y_Lift : FB_Cylinder;
	Index03_Y_Stopper : FB_Cylinder;
	Index04_B_Detect : FB_SensorBinary;
	Index04_B_Exit : FB_SensorBinary;
	Index04_Y_Lift : FB_Cylinder;
	Index04_Y_Stopper : FB_Cylinder;
	Index05_B_Detect : FB_SensorBinary;
	Index05_B_Exit : FB_SensorBinary;
	Index05_Y_Lift : FB_Cylinder;
	Index05_Y_Stopper : FB_Cylinder;
	Lift01_B_Detect : FB_SensorBinary;
	Lift01_B_Exit : FB_SensorBinary;
	Lift01_M_Conveyor : FB_Drive;
	Lift01_Y_Lift : FB_Cylinder;
	Lift02_B_Detect : FB_SensorBinary;
	Lift02_B_Exit : FB_SensorBinary;
	Lift02_M_Conveyor : FB_Drive;
	Lift02_Y_Lift : FB_Cylinder;
	Stopper01_B_Detect : FB_SensorBinary;
	Stopper01_B_Exit : FB_SensorBinary;
	Stopper01_Y_Stopper : FB_Cylinder;
	Stopper02_B_Detect : FB_SensorBinary;
	Stopper02_B_Exit : FB_SensorBinary;
	Stopper02_Y_Stopper : FB_Cylinder;
	Stopper03_B_Detect : FB_SensorBinary;
	Stopper03_B_Exit : FB_SensorBinary;
	Stopper03_Y_Stopper : FB_Cylinder;
	Stopper04_B_Detect : FB_SensorBinary;
	Stopper04_B_Exit : FB_SensorBinary;
	Stopper04_Y_Stopper : FB_Cylinder;
	Transport01_M_Conveyor : FB_Drive;
	Transport02_M_Conveyor : FB_Drive;
END_VAR
{endregion}

{region generated code}
	InitRun();
	Index01_B_Detect();
	Index01_B_Exit();
	Index01_Y_Lift();
	Index01_Y_Stopper();
	Index02_B_Detect();
	Index02_B_Exit();
	Index02_Y_Lift();
	Index02_Y_Stopper();
	Index03_B_Detect();
	Index03_B_Exit();
	Index03_Y_Lift();
	Index03_Y_Stopper();
	Index04_B_Detect();
	Index04_B_Exit();
	Index04_Y_Lift();
	Index04_Y_Stopper();
	Index05_B_Detect();
	Index05_B_Exit();
	Index05_Y_Lift();
	Index05_Y_Stopper();
	Lift01_B_Detect();
	Lift01_B_Exit();
	Lift01_M_Conveyor();
	Lift01_Y_Lift();
	Lift02_B_Detect();
	Lift02_B_Exit();
	Lift02_M_Conveyor();
	Lift02_Y_Lift();
	Stopper01_B_Detect();
	Stopper01_B_Exit();
	Stopper01_Y_Stopper();
	Stopper02_B_Detect();
	Stopper02_B_Exit();
	Stopper02_Y_Stopper();
	Stopper03_B_Detect();
	Stopper03_B_Exit();
	Stopper03_Y_Stopper();
	Stopper04_B_Detect();
	Stopper04_B_Exit();
	Stopper04_Y_Stopper();
	Transport01_M_Conveyor();
	Transport02_M_Conveyor();
{endregion}

Mapping();

METHOD InitRun
{region generated code}
VAR_INST
	bInitRun : BOOL := TRUE;
END_VAR
{endregion}
{region generated code}
	IF NOT bInitRun THEN RETURN; END_IF
	bInitRun := FALSE;
{endregion}
END_METHOD

ACTION Mapping:
// ============================================================================
// FG_Transport twin <-> PLCSIM Advanced process image.
//
// Addresses: Siemens/_data/PLCTags_FG_Transport.xlsx.
//
// One byte per station, in the table's own order: Index01..05 on %I/%Q1003..1007,
// Stopper01..04 on 1008..1011, Lift01/02 on 1012/1013, Transport01/02 on
// 1014/1015. The bit positions repeat exactly per station type, so read one
// block and you have read them all.
//
// THE TWO GATES ARE NOT MAPPED HERE ANY MORE. FG_TS_Gate_1 / _2 keep their
// %I1001 / %I1002 addresses in this table, but the twin devices Y_Gate1 and
// Y_Gate2 live in FG_01 now - they are not members of this function block and
// assigning them here did not compile. They are mapped in FG_01's Mapping action,
// from these same addresses.
//
// Three things that are easy to get backwards:
//
//   * A STOPPER IS RETRACTED WHEN IT HOLDS THE PALLET. InHome %I1xxx.4 is
//     "Stopper geschlossen" and WorkPos %Q1xxx.2 is "Stopper oeffnen" - so
//     EXTENDING RELEASES. Nine authored Function entries in the twin say the
//     opposite and are known to be wrong; the table agrees with reality, not
//     with the twin's prose.
//   * A LIFT IS RETRACTED WHEN IT IS DOWN. InHome "Heber ist unten",
//     HomePos "Heber senken".
//   * ON A DRIVE, nControl.0 IS FORWARDS AND nControl.1 IS BACKWARDS. The table
//     names them: _Plus is "Antrieb vorwaerts", _Minus is "Antrieb rueckwaerts",
//     and Plus is always the LOWER address of the pair. THE PREVIOUS MAPPING HAD
//     ALL FOUR DRIVES INVERTED - it copied the Beckhoff side's channel order,
//     where the lower channel happens to be nControl.1, onto Siemens addresses
//     where the lower address is Plus. Every belt ran the wrong way.
// ============================================================================

// --- Index01 - detect, exit, lift and stopper on byte 1003 --------------
GVL_PLC.Inputs.I1003.0	:= Index01_B_Detect.bValue;
GVL_PLC.Inputs.I1003.1	:= Index01_B_Exit.bValue;
GVL_PLC.Inputs.I1003.2	:= Index01_Y_Lift.bRetracted;		// "Heber ist unten"
GVL_PLC.Inputs.I1003.3	:= Index01_Y_Lift.bExtended;		// "Heber ist oben"
GVL_PLC.Inputs.I1003.4	:= Index01_Y_Stopper.bRetracted;		// "Stopper geschlossen"
Index01_Y_Lift.bRetract	:= GVL_PLC.Outputs.Q1003.0;		// "Heber senken"
Index01_Y_Lift.bExtend	:= GVL_PLC.Outputs.Q1003.1;		// "Heber heben"
Index01_Y_Stopper.bExtend	:= GVL_PLC.Outputs.Q1003.2;		// "Stopper oeffnen"

// --- Index02 - detect, exit, lift and stopper on byte 1004 --------------
GVL_PLC.Inputs.I1004.0	:= Index02_B_Detect.bValue;
GVL_PLC.Inputs.I1004.1	:= Index02_B_Exit.bValue;
GVL_PLC.Inputs.I1004.2	:= Index02_Y_Lift.bRetracted;		// "Heber ist unten"
GVL_PLC.Inputs.I1004.3	:= Index02_Y_Lift.bExtended;		// "Heber ist oben"
GVL_PLC.Inputs.I1004.4	:= Index02_Y_Stopper.bRetracted;		// "Stopper geschlossen"
Index02_Y_Lift.bRetract	:= GVL_PLC.Outputs.Q1004.0;		// "Heber senken"
Index02_Y_Lift.bExtend	:= GVL_PLC.Outputs.Q1004.1;		// "Heber heben"
Index02_Y_Stopper.bExtend	:= GVL_PLC.Outputs.Q1004.2;		// "Stopper oeffnen"

// --- Index03 - detect, exit, lift and stopper on byte 1005 --------------
GVL_PLC.Inputs.I1005.0	:= Index03_B_Detect.bValue;
GVL_PLC.Inputs.I1005.1	:= Index03_B_Exit.bValue;
GVL_PLC.Inputs.I1005.2	:= Index03_Y_Lift.bRetracted;		// "Heber ist unten"
GVL_PLC.Inputs.I1005.3	:= Index03_Y_Lift.bExtended;		// "Heber ist oben"
GVL_PLC.Inputs.I1005.4	:= Index03_Y_Stopper.bRetracted;		// "Stopper geschlossen"
Index03_Y_Lift.bRetract	:= GVL_PLC.Outputs.Q1005.0;		// "Heber senken"
Index03_Y_Lift.bExtend	:= GVL_PLC.Outputs.Q1005.1;		// "Heber heben"
Index03_Y_Stopper.bExtend	:= GVL_PLC.Outputs.Q1005.2;		// "Stopper oeffnen"

// --- Index04 - detect, exit, lift and stopper on byte 1006 --------------
GVL_PLC.Inputs.I1006.0	:= Index04_B_Detect.bValue;
GVL_PLC.Inputs.I1006.1	:= Index04_B_Exit.bValue;
GVL_PLC.Inputs.I1006.2	:= Index04_Y_Lift.bRetracted;		// "Heber ist unten"
GVL_PLC.Inputs.I1006.3	:= Index04_Y_Lift.bExtended;		// "Heber ist oben"
GVL_PLC.Inputs.I1006.4	:= Index04_Y_Stopper.bRetracted;		// "Stopper geschlossen"
Index04_Y_Lift.bRetract	:= GVL_PLC.Outputs.Q1006.0;		// "Heber senken"
Index04_Y_Lift.bExtend	:= GVL_PLC.Outputs.Q1006.1;		// "Heber heben"
Index04_Y_Stopper.bExtend	:= GVL_PLC.Outputs.Q1006.2;		// "Stopper oeffnen"

// --- Index05 - detect, exit, lift and stopper on byte 1007 --------------
GVL_PLC.Inputs.I1007.0	:= Index05_B_Detect.bValue;
GVL_PLC.Inputs.I1007.1	:= Index05_B_Exit.bValue;
GVL_PLC.Inputs.I1007.2	:= Index05_Y_Lift.bRetracted;		// "Heber ist unten"
GVL_PLC.Inputs.I1007.3	:= Index05_Y_Lift.bExtended;		// "Heber ist oben"
GVL_PLC.Inputs.I1007.4	:= Index05_Y_Stopper.bRetracted;		// "Stopper geschlossen"
Index05_Y_Lift.bRetract	:= GVL_PLC.Outputs.Q1007.0;		// "Heber senken"
Index05_Y_Lift.bExtend	:= GVL_PLC.Outputs.Q1007.1;		// "Heber heben"
Index05_Y_Stopper.bExtend	:= GVL_PLC.Outputs.Q1007.2;		// "Stopper oeffnen"

// --- Stopper01 - detect, exit and stopper on byte 1008 --------------------
GVL_PLC.Inputs.I1008.0	:= Stopper01_B_Detect.bValue;
GVL_PLC.Inputs.I1008.1	:= Stopper01_B_Exit.bValue;
GVL_PLC.Inputs.I1008.4	:= Stopper01_Y_Stopper.bRetracted;		// "Stopper geschlossen"
Stopper01_Y_Stopper.bExtend	:= GVL_PLC.Outputs.Q1008.2;		// "Stopper oeffnen"

// --- Stopper02 - detect, exit and stopper on byte 1009 --------------------
GVL_PLC.Inputs.I1009.0	:= Stopper02_B_Detect.bValue;
GVL_PLC.Inputs.I1009.1	:= Stopper02_B_Exit.bValue;
GVL_PLC.Inputs.I1009.4	:= Stopper02_Y_Stopper.bRetracted;		// "Stopper geschlossen"
Stopper02_Y_Stopper.bExtend	:= GVL_PLC.Outputs.Q1009.2;		// "Stopper oeffnen"

// --- Stopper03 - detect, exit and stopper on byte 1010 --------------------
GVL_PLC.Inputs.I1010.0	:= Stopper03_B_Detect.bValue;
GVL_PLC.Inputs.I1010.1	:= Stopper03_B_Exit.bValue;
GVL_PLC.Inputs.I1010.4	:= Stopper03_Y_Stopper.bRetracted;		// "Stopper geschlossen"
Stopper03_Y_Stopper.bExtend	:= GVL_PLC.Outputs.Q1010.2;		// "Stopper oeffnen"

// --- Stopper04 - detect, exit and stopper on byte 1011 --------------------
GVL_PLC.Inputs.I1011.0	:= Stopper04_B_Detect.bValue;
GVL_PLC.Inputs.I1011.1	:= Stopper04_B_Exit.bValue;
GVL_PLC.Inputs.I1011.4	:= Stopper04_Y_Stopper.bRetracted;		// "Stopper geschlossen"
Stopper04_Y_Stopper.bExtend	:= GVL_PLC.Outputs.Q1011.2;		// "Stopper oeffnen"

// --- Lift01 - detect, exit, lift and carriage belt on byte 1012 --------
GVL_PLC.Inputs.I1012.0	:= Lift01_B_Detect.bValue;
GVL_PLC.Inputs.I1012.1	:= Lift01_B_Exit.bValue;
GVL_PLC.Inputs.I1012.2	:= Lift01_Y_Lift.bRetracted;		// "Heber ist unten"
GVL_PLC.Inputs.I1012.3	:= Lift01_Y_Lift.bExtended;		// "Heber ist oben"
Lift01_Y_Lift.bRetract	:= GVL_PLC.Outputs.Q1012.0;		// "Heber senken"
Lift01_Y_Lift.bExtend	:= GVL_PLC.Outputs.Q1012.1;		// "Heber heben"
Lift01_M_Conveyor.nControl.0	:= GVL_PLC.Outputs.Q1012.2;		// _Plus  "Antrieb vorwaerts"
Lift01_M_Conveyor.nControl.1	:= GVL_PLC.Outputs.Q1012.3;		// _Minus "Antrieb rueckwaerts"

// --- Lift02 - detect, exit, lift and carriage belt on byte 1013 --------
GVL_PLC.Inputs.I1013.0	:= Lift02_B_Detect.bValue;
GVL_PLC.Inputs.I1013.1	:= Lift02_B_Exit.bValue;
GVL_PLC.Inputs.I1013.2	:= Lift02_Y_Lift.bRetracted;		// "Heber ist unten"
GVL_PLC.Inputs.I1013.3	:= Lift02_Y_Lift.bExtended;		// "Heber ist oben"
Lift02_Y_Lift.bRetract	:= GVL_PLC.Outputs.Q1013.0;		// "Heber senken"
Lift02_Y_Lift.bExtend	:= GVL_PLC.Outputs.Q1013.1;		// "Heber heben"
Lift02_M_Conveyor.nControl.0	:= GVL_PLC.Outputs.Q1013.2;		// _Plus  "Antrieb vorwaerts"
Lift02_M_Conveyor.nControl.1	:= GVL_PLC.Outputs.Q1013.3;		// _Minus "Antrieb rueckwaerts"

// --- Transport01 - the level 1 circulation belt, byte 1014 -------------------
Transport01_M_Conveyor.nControl.0	:= GVL_PLC.Outputs.Q1014.0;		// _Plus  "Antrieb vorwaerts"
Transport01_M_Conveyor.nControl.1	:= GVL_PLC.Outputs.Q1014.1;		// _Minus "Antrieb rueckwaerts"

// --- Transport02 - the level 2 circulation belt, byte 1015 -------------------
Transport02_M_Conveyor.nControl.0	:= GVL_PLC.Outputs.Q1015.0;		// _Plus  "Antrieb vorwaerts"
Transport02_M_Conveyor.nControl.1	:= GVL_PLC.Outputs.Q1015.1;		// _Minus "Antrieb rueckwaerts"

// TODO: NO INPUT ADDRESS IN PLCTags_FG_Transport.xlsx for ANY of the four drives'
// running feedback. Every FB_Drive publishes nStatus.6 - "moving", written every
// scan - and none of the four has a tag for it, so the control PLC commands a belt
// and is never told whether it turned. A running belt is not a moving pallet, but
// a belt that never started is not either, and today the PLC cannot tell those
// apart. Add four input bits:
//   GVL_PLC.Inputs.I<n>.<b> := Lift01_M_Conveyor.nStatus.6;
//   GVL_PLC.Inputs.I<n>.<b> := Lift02_M_Conveyor.nStatus.6;
//   GVL_PLC.Inputs.I<n>.<b> := Transport01_M_Conveyor.nStatus.6;
//   GVL_PLC.Inputs.I<n>.<b> := Transport02_M_Conveyor.nStatus.6;
// nStatus.7 is NOT a health bit - it is a one second init pulse. Do not map it.

// TODO: NO Y_Stopper_InWork IN THE TABLE for any of the nine stoppers. Only the
// closed limit is published, so .bExtended goes nowhere and the PLC can see that
// a stopper has left the blocking position but never that it is fully clear. The
// Beckhoff side reads both limits on every stopper. Add %I1xxx.5 per station.
END_ACTION

END_FUNCTION_BLOCK
